    10:
        IF THIS^.WriteGCodeFile('TangentialCut.nc') THEN
            ADSLOGSTR(ADSLOG_MSGTYPE_HINT, 'Generator: Zapisano plik TangentialCut.nc', '');
            nBuildStep := 1000;
        END_IF

    1000:
        _Busy := FALSE;
        _Done := TRUE; 
        nBuildStep := 0;
        Build := TRUE;
        
END_CASE
END_METHOD

METHOD PROTECTED CalculateFootprint
VAR_INPUT
END_VAR
_NominalX := _Config.Diameter;
_NominalY := _Config.Diameter;
END_METHOD

PROPERTY ExecutionRoute : E_ExecutionRoute
GET
ExecutionRoute := E_ExecutionRoute.eGCode;
END_GET
END_PROPERTY

METHOD FB_init : BOOL
VAR_INPUT
	bInitRetains : BOOL; // if TRUE, the retain variables are initialized (warm start / cold start)
	bInCopyCode : BOOL;  // if TRUE, the instance afterwards gets moved into the copy code (online change)
END_VAR
_Limits.PanelFrontLength.MinVal := 100.0;
_Limits.PanelFrontLength.MaxVal := 2400.0;

_Limits.PanelFrontWidth.MinVal  := 100.0;
_Limits.PanelFrontWidth.MaxVal  := 1200.0;

_Limits.PanelHeight.MinVal      := 0.0;
_Limits.PanelHeight.MaxVal      := 0.0;

_Limits.RailHeightCorrection.MinVal := 0.0;
_Limits.RailHeightCorrection.MaxVal := 0.0;

_Limits.CuttingOverpass.MinVal := 0.0;
_Limits.CuttingOverpass.MaxVal := 50.0;

_Limits.GroovingOverpass.MinVal := 0.0;
_Limits.GroovingOverpass.MaxVal := 50.0;

_Limits.GrooveDepthZ.MinVal := 0.0;
_Limits.GrooveDepthZ.MaxVal := 9.0; 

_Limits.Diameter.MinVal := 10;
_Limits.Diameter.MaxVal := 600;
END_METHOD

END_FUNCTION_BLOCK

// ---- POUs/Builder/Recipes/FB_FeedRoundedRectangle.TcPOU
FUNCTION_BLOCK FB_FeedRoundedRectangle EXTENDS FB_RecipeBase

METHOD Build : BOOL
VAR
    TotalX, TotalY, Radius : LREAL;
    Velo : LREAL;
    localConfig : ST_GantryXYZ_Config;
	SmallRadius : LREAL;
    SmallMinX   : LREAL;
    SmallMaxX   : LREAL;
    SmallMinY   : LREAL;
    SmallMaxY   : LREAL;
END_VAR
_Busy := TRUE;
_Done := FALSE;
_Error := FALSE;
Build := FALSE;
THIS^.UpdateNestingLimits();

IF NOT _Config.IsValid THEN
    _Busy := FALSE;
    _Error := TRUE; 
    Build := FALSE;
    RETURN;
END_IF

// Gabaryty i promień
TotalX := _Config.PanelFrontWidth;
TotalY := _Config.PanelFrontLength;
Radius := _Config.Radius;

IF Radius > (TotalX / 2.0) THEN Radius := TotalX / 2.0; END_IF
IF Radius > (TotalY / 2.0) THEN Radius := TotalY / 2.0; END_IF

IF _ConfigProvider <> 0 THEN
    localConfig := _ConfigProvider.Config;
    Velo := localConfig.CuttingSpeedXY;
ELSE
    Velo := 50.0;
END_IF

// ===================================================
// DEFINICJA ILOŚCI I PUNKTÓW STARTOWYCH
// ===================================================
_ShapesCount := 1; 

// Kształt 1: Zewnętrzny prostokąt (100%) - Zaczynamy na środku PRAWEJ krawędzi
_ShapeStart[1].X := TotalX;
_ShapeStart[1].Y := TotalY / 2.0;

// Obliczenia dla małego prostokąta (50% wielkości, wyśrodkowany)
SmallMinX := TotalX * 0.25;
SmallMaxX := TotalX * 0.75;
SmallMinY := TotalY * 0.25;
SmallMaxY := TotalY * 0.75;
SmallRadius := Radius * 0.5;

// Kształt 2: Wewnętrzny prostokąt (50%) - Zaczynamy na środku PRAWEJ krawędzi
_ShapeStart[2].X := SmallMaxX;
_ShapeStart[2].Y := TotalY / 2.0;


// ============================================
// GENEROWANIE TABELI (Ruch CCW / Lewoskrętnie)
// ============================================
_GeometryWriter.Clear();
_GeometryWriter.EnableTangentialFollowing();

CASE _CurrentShapeIndex OF
    1:
        // ----------------------------------------------------
        // RYSOWANIE DUŻEGO PROSTOKĄTA (KSZTAŁT 1)
        // ----------------------------------------------------
        _GeometryWriter.AddStartPoint(_ShapeStart[1].X, _ShapeStart[1].Y);

        // 1. Prawa krawędź -> Prawy górny łuk (Tniemy w +Y, Q = 0)
        _GeometryWriter.AddLine(TotalX, TotalY - Radius, Velo);
        IF Radius > 0 THEN
            // FALSE = G03 = CounterClockwise (Lewoskrętnie)
            _GeometryWriter.AddArc(TotalX - Radius, TotalY, TotalX - Radius, TotalY - Radius, Velo, FALSE);
        END_IF

        // 2. Górna krawędź -> Lewy górny łuk (Tniemy w -X, Q = 90)
        _GeometryWriter.AddLine(Radius, TotalY, Velo);
        IF Radius > 0 THEN
            _GeometryWriter.AddArc(0.0, TotalY - Radius, Radius, TotalY - Radius, Velo, FALSE);
        END_IF

        // 3. Lewa krawędź -> Lewy dolny łuk (Tniemy w -Y, Q = 180)
        _GeometryWriter.AddLine(0.0, Radius, Velo);
        IF Radius > 0 THEN
            _GeometryWriter.AddArc(Radius, 0.0, Radius, Radius, Velo, FALSE);
        END_IF

        // 4. Dolna krawędź -> Prawy dolny łuk (Tniemy w +X, Q = 270)
        _GeometryWriter.AddLine(TotalX - Radius, 0.0, Velo);
        IF Radius > 0 THEN
            _GeometryWriter.AddArc(TotalX, Radius, TotalX - Radius, Radius, Velo, FALSE);
        END_IF

        // Zamknięcie na prawej krawędzi
        _GeometryWriter.AddLine(TotalX, TotalY / 2.0, Velo);

END_CASE

_GeometryWriter.EndTable();

_Busy := FALSE;
_Done := TRUE;
Build := TRUE;
END_METHOD

METHOD PROTECTED CalculateFootprint
VAR_INPUT
END_VAR
_NominalX := _Config.PanelFrontWidth;
_NominalY := _Config.PanelFrontLength;
END_METHOD

PROPERTY ExecutionRoute : E_ExecutionRoute
GET
ExecutionRoute := E_ExecutionRoute.eFeedTable;
END_GET
END_PROPERTY

METHOD FB_init : BOOL
VAR_INPUT
	bInitRetains : BOOL; // if TRUE, the retain variables are initialized (warm start / cold start)
	bInCopyCode : BOOL;  // if TRUE, the instance afterwards gets moved into the copy code (online change)
END_VAR
_Limits.PanelFrontLength.MinVal := 50.0;
_Limits.PanelFrontLength.MaxVal := 2400.0;

_Limits.PanelFrontWidth.MinVal  := 50.0;
_Limits.PanelFrontWidth.MaxVal  := 1200.0;

_Limits.PanelHeight.MinVal      := 0.0;
_Limits.PanelHeight.MaxVal      := 0.0;

_Limits.RailHeightCorrection.MinVal := 0.0;
_Limits.RailHeightCorrection.MaxVal := 0.0;

_Limits.CuttingOverpass.MinVal := 0.0;
_Limits.CuttingOverpass.MaxVal := 50.0;

_Limits.GroovingOverpass.MinVal := 0.0;
_Limits.GroovingOverpass.MaxVal := 50.0;

_Limits.GrooveDepthZ.MinVal := 0.0;
_Limits.GrooveDepthZ.MaxVal := 9.0; 

_Limits.CuttingOverpass.MinVal := 0.0;
_Limits.CuttingOverpass.MaxVal := 50.0;
_Limits.GroovingOverpass.MinVal := 0.0;
_Limits.GroovingOverpass.MaxVal := 50.0;

_Limits.Radius.MinVal := 10.0;     
_Limits.Radius.MaxVal := 600.0;
END_METHOD

END_FUNCTION_BLOCK

// ---- POUs/Builder/Recipes/FB_FeedCircle.TcPOU
FUNCTION_BLOCK FB_FeedCircle EXTENDS FB_RecipeBase

METHOD Build : BOOL
VAR
    TotalX, Radius : LREAL;
    Velo : LREAL;
    localConfig : ST_GantryXYZ_Config;
    LeadInY : LREAL := 20.0;
    LeadOutY : LREAL := 20.0;
END_VAR
_Busy := TRUE;
_Done := FALSE;
_Error := FALSE;
Build := FALSE;

THIS^.UpdateNestingLimits();

IF NOT _Config.IsValid THEN
    _Busy := FALSE;
    _Error := TRUE;
    RETURN;
END_IF

TotalX := _Config.Diameter;
Radius := TotalX / 2.0;

// ===================================================
// DEFINICJA ILOŚCI I PUNKTÓW STARTOWYCH
// ===================================================
_ShapesCount := 1; 

_ShapeStart[1].X := TotalX;
_ShapeStart[1].Y := Radius - LeadInY;

IF _ConfigProvider <> 0 THEN
    localConfig := _ConfigProvider.Config;
    Velo := localConfig.CuttingSpeedXY;
ELSE
    Velo := 50.0;
END_IF

_GeometryWriter.Clear();
_GeometryWriter.EnableTangentialFollowing();

// RYSOWANIE TYLKO TEGO KSZTAŁTU, O KTÓRY PROSI EXECUTOR
CASE _CurrentShapeIndex OF
    1:
        _GeometryWriter.AddStartPoint(_ShapeStart[1].X, _ShapeStart[1].Y); 
        _GeometryWriter.AddLine(TotalX, Radius, Velo); 
        _GeometryWriter.AddArc(0.0, Radius, Radius, Radius, Velo, FALSE);
        _GeometryWriter.AddArc(TotalX, Radius, Radius, Radius, Velo, FALSE);
        _GeometryWriter.AddLine(TotalX, Radius + LeadOutY, Velo); 
END_CASE

_GeometryWriter.EndTable();

_Busy := FALSE;
_Done := TRUE;
Build := TRUE;
END_METHOD

METHOD PROTECTED CalculateFootprint
VAR_INPUT
END_VAR
_NominalX := _Config.Diameter;
_NominalY := _Config.Diameter;
END_METHOD

PROPERTY ExecutionRoute : E_ExecutionRoute
GET
ExecutionRoute := E_ExecutionRoute.eFeedTable;
END_GET
END_PROPERTY

METHOD FB_init : BOOL
VAR_INPUT
	bInitRetains : BOOL; // if TRUE, the retain variables are initialized (warm start / cold start)
	bInCopyCode : BOOL;  // if TRUE, the instance afterwards gets moved into the copy code (online change)
END_VAR
_Limits.Diameter.MinVal := 50.0;
_Limits.Diameter.MaxVal := 1200.0;
_Limits.Radius.MinVal := 10.0;
_Limits.Radius.MaxVal := 100;

_Limits.CuttingOverpass.MinVal := 0.0;
_Limits.CuttingOverpass.MaxVal := 50.0;
_Limits.GroovingOverpass.MinVal := 0.0;
_Limits.GroovingOverpass.MaxVal := 50.0;
END_METHOD

END_FUNCTION_BLOCK

// ---- POUs/Builder/Recipes/FB_FeedMeina2_2000x1000.TcPOU
FUNCTION_BLOCK FB_FeedMeina2_2000x1000 EXTENDS FB_RecipeBase

METHOD Build : BOOL
VAR
    TotalX, TotalY, Radius : LREAL;
    Velo : LREAL;
    localConfig : ST_GantryXYZ_Config;
	
    // Zmienne do otworów
    HoleDistanceFromEdgeOfRail : LREAL := 100.0;
    SomeFixedDimension         : LREAL := 12.63;
    PanelRailOffsetX           : LREAL;
    PanelRailOffsetY           : LREAL;
    ExtrusionLengthX           : LREAL;
    ExtrusionLengthY           : LREAL;
    
    NumberOfHolesX             : INT := 3;
    NumberOfHolesY             : INT := 5;
    HolesSpacingX              : LREAL;
    HolesSpacingY              : LREAL;
    
    i                          : INT;
    holeIdx                    : INT;
	
	RailSlot  : LREAL := 29.0;
	BigSlot   : LREAL := 200.0;
	SmallSlot : LREAL := 100.0;

// Zmienne pomocnicze do generowania ścieżek
	sx : LREAL;
	sy : LREAL;
	dx : LREAL;
	dy : LREAL;
	r_val : LREAL;
	
END_VAR
_Busy := TRUE;
_Done := FALSE;
_Error := FALSE;
Build := FALSE;
THIS^.UpdateNestingLimits();

IF NOT _Config.IsValid THEN
    _Busy := FALSE;
    _Error := TRUE; 
    Build := FALSE;
    RETURN;
END_IF

// Gabaryty i promień
TotalX := 1000;
TotalY := 2000;
Radius := _Config.Radius;

IF Radius > (TotalX / 2.0) THEN Radius := TotalX / 2.0; END_IF
IF Radius > (TotalY / 2.0) THEN Radius := TotalY / 2.0; END_IF


// ===================================================
// OBLICZENIA DLA SZYN I OTWORÓW
// ===================================================
// Po poprawce: offset X uzależniony od X, a Y od Y
PanelRailOffsetX := 0.1 * TotalX;
PanelRailOffsetY := 0.1 * TotalY;

ExtrusionLengthX := TotalX - (2.0 * PanelRailOffsetX);
ExtrusionLengthY := TotalY - (2.0 * PanelRailOffsetY);

// Wyliczenie rozstawu (Zabezpieczenie przed dzieleniem przez zero, jeśli ktoś wpisze NumberOfHoles = 1)
IF NumberOfHolesX > 1 THEN
    HolesSpacingX := (ExtrusionLengthX - (2.0 * HoleDistanceFromEdgeOfRail)) / INT_TO_LREAL(NumberOfHolesX - 1);
ELSE
    HolesSpacingX := 0.0;
END_IF

IF NumberOfHolesY > 1 THEN
    HolesSpacingY := (ExtrusionLengthY - (2.0 * HoleDistanceFromEdgeOfRail)) / INT_TO_LREAL(NumberOfHolesY - 1);
ELSE
    HolesSpacingY := 0.0;
END_IF


// ===================================================
// GENEROWANIE OTWORÓW (Zoptymalizowana ścieżka po obwodzie)
// ===================================================
holeIdx := 1;

// 1. Otwór na dokładnym środku wycinanego detalu
_HolesDrill[holeIdx].X := LREAL_TO_REAL(TotalX / 2.0);
_HolesDrill[holeIdx].Y := LREAL_TO_REAL(TotalY / 2.0);

// 2. Rail Y1 (Lewa) - Ruch z GÓRY na DÓŁ
FOR i := NumberOfHolesY TO 1 BY -1 DO
    holeIdx := holeIdx + 1;
    _HolesDrill[holeIdx].X := LREAL_TO_REAL(PanelRailOffsetX - SomeFixedDimension);
    _HolesDrill[holeIdx].Y := LREAL_TO_REAL(PanelRailOffsetY + HoleDistanceFromEdgeOfRail + ((i - 1) * HolesSpacingY));
END_FOR

// 3. Rail X1 (Dolna) - Ruch z LEWEJ do PRAWEJ
FOR i := 1 TO NumberOfHolesX DO
    holeIdx := holeIdx + 1;
    _HolesDrill[holeIdx].X := LREAL_TO_REAL(PanelRailOffsetX + HoleDistanceFromEdgeOfRail + ((i - 1) * HolesSpacingX));
    _HolesDrill[holeIdx].Y := LREAL_TO_REAL(PanelRailOffsetY - SomeFixedDimension);
END_FOR

// 4. Rail Y2 (Prawa) - Ruch z DOŁU do GÓRY
FOR i := 1 TO NumberOfHolesY DO
    holeIdx := holeIdx + 1;
    _HolesDrill[holeIdx].X := LREAL_TO_REAL(PanelRailOffsetX + ExtrusionLengthX + SomeFixedDimension);
    _HolesDrill[holeIdx].Y := LREAL_TO_REAL(PanelRailOffsetY + HoleDistanceFromEdgeOfRail + ((i - 1) * HolesSpacingY));
END_FOR

// 5. Rail X2 (Górna) - Ruch z PRAWEJ do LEWEJ
FOR i := NumberOfHolesX TO 1 BY -1 DO
    holeIdx := holeIdx + 1;
    _HolesDrill[holeIdx].X := LREAL_TO_REAL(PanelRailOffsetX + HoleDistanceFromEdgeOfRail + ((i - 1) * HolesSpacingX));
    _HolesDrill[holeIdx].Y := LREAL_TO_REAL(PanelRailOffsetY + ExtrusionLengthY + SomeFixedDimension);
END_FOR

// Przypisanie całkowitej liczby otworów do recepty
_HolesToDrill := holeIdx;

// ===================================================
// DEFINICJA ILOŚCI I PUNKTÓW STARTOWYCH (Dla FeedTable)
// ===================================================
_ShapesCount := 6; // 1 główny panel + 5 nowych wycięć z tabeli

// 1. Kształt główny
_ShapeStart[1].X := 0.0;
_ShapeStart[1].Y := 0.0;

// 2. No. 1
_ShapeStart[2].X := 1030.0;
_ShapeStart[2].Y := 0.0;

// 3. No. 2
_ShapeStart[3].X := 1090.0;
_ShapeStart[3].Y := 0.0;

// 4. No. 3
_ShapeStart[4].X := 210.0;
_ShapeStart[4].Y := 2200.0;

// 5. No. 4
_ShapeStart[5].X := 410.0;
_ShapeStart[5].Y := 2150.0;

// 6. No. 5
_ShapeStart[6].X := 810.0;
_ShapeStart[6].Y := 2150.0;

IF _ConfigProvider <> 0 THEN
    localConfig := _ConfigProvider.Config;
    Velo := localConfig.CuttingSpeedXY;
ELSE
    Velo := 50.0;
END_IF

_GeometryWriter.Clear();
_GeometryWriter.EnableTangentialFollowing();

// Reset zmiennych pomocniczych przed każdym wywołaniem
sx := 0.0; sy := 0.0; dx := 0.0; dy := 0.0; r_val := 0.0;

// RYSOWANIE KSZTAŁTU ZGODNIE Z INDEKSEM
CASE _CurrentShapeIndex OF
    1:
        // ==========================================
        // KSZTAŁT 1 (Główny panel - Twój stary kod)
        // ==========================================
        _GeometryWriter.AddStartPoint(_ShapeStart[1].X, _ShapeStart[1].Y);

        _GeometryWriter.AddLine(0.0, TotalY - Radius, Velo);
        IF Radius > 0 THEN
            _GeometryWriter.AddArc(Radius, TotalY, Radius, TotalY - Radius, Velo, TRUE);
        END_IF

        _GeometryWriter.AddLine(TotalX - Radius, TotalY, Velo);
        IF Radius > 0 THEN
            _GeometryWriter.AddArc(TotalX, TotalY - Radius, TotalX - Radius, TotalY - Radius, Velo, TRUE);
        END_IF

        _GeometryWriter.AddLine(TotalX, Radius, Velo);
        IF Radius > 0 THEN
            _GeometryWriter.AddArc(TotalX - Radius, 0.0, TotalX - Radius, Radius, Velo, TRUE);
        END_IF

        _GeometryWriter.AddLine(Radius, 0.0, Velo);
        IF Radius > 0 THEN
            _GeometryWriter.AddArc(0.0, Radius, Radius, Radius, Velo, TRUE);
        END_IF

    2, 3, 4, 5, 6:
        // ==========================================
        // KSZTAŁTY OD 2 DO 6 (Z tabeli)
        // ==========================================
        // Przypisanie współrzędnych startowych dla aktualnego kształtu
        sx := _ShapeStart[_CurrentShapeIndex].X;
        sy := _ShapeStart[_CurrentShapeIndex].Y;
        r_val := 10.0; // Promień jest równy 10 dla wszystkich slotów

        // Dobór wymiarów na podstawie tego, który numer wycinamy
        IF _CurrentShapeIndex = 2 THEN
            dx := RailSlot;
            dy := ExtrusionLengthY;
        ELSIF _CurrentShapeIndex = 3 THEN
            dx := RailSlot;
            dy := ExtrusionLengthX;
        ELSIF _CurrentShapeIndex = 4 THEN
            dx := SmallSlot;
            dy := SmallSlot;
        ELSIF _CurrentShapeIndex = 5 THEN
            dx := BigSlot;
            dy := BigSlot;
        ELSIF _CurrentShapeIndex = 6 THEN
            dx := BigSlot;
            dy := BigSlot;
        END_IF

        // Wygenerowanie geometrycznej ścieżki (z absolutnym offsetem sx, sy)
        // Wkłuwamy się w lewym dolnym rogu (w odpad)
        _GeometryWriter.AddStartPoint(sx, sy);

        // 1. Lewa krawędź w górę
        _GeometryWriter.AddLine(sx, sy + dy - r_val, Velo);
        IF r_val > 0 THEN
            // Lewy górny łuk
            _GeometryWriter.AddArc(sx + r_val, sy + dy, sx + r_val, sy + dy - r_val, Velo, TRUE);
        END_IF

        // 2. Górna krawędź w prawo
        _GeometryWriter.AddLine(sx + dx - r_val, sy + dy, Velo);
        IF r_val > 0 THEN
            // Prawy górny łuk
            _GeometryWriter.AddArc(sx + dx, sy + dy - r_val, sx + dx - r_val, sy + dy - r_val, Velo, TRUE);
        END_IF

        // 3. Prawa krawędź w dół
        _GeometryWriter.AddLine(sx + dx, sy + r_val, Velo);
        IF r_val > 0 THEN
            // Prawy dolny łuk
            _GeometryWriter.AddArc(sx + dx - r_val, sy, sx + dx - r_val, sy + r_val, Velo, TRUE);
        END_IF

        // 4. Dolna krawędź w lewo i zamknięcie
        _GeometryWriter.AddLine(sx + r_val, sy, Velo);
        IF r_val > 0 THEN
            // Lewy dolny łuk
            _GeometryWriter.AddArc(sx, sy + r_val, sx + r_val, sy + r_val, Velo, TRUE);
        END_IF

END_CASE

_GeometryWriter.EndTable();

_Busy := FALSE;
_Done := TRUE;
Build := TRUE;
END_METHOD

METHOD PROTECTED CalculateFootprint
VAR_INPUT
END_VAR
_NominalX := 1200;
_NominalY := 2400;
END_METHOD

PROPERTY ExecutionRoute : E_ExecutionRoute
GET
ExecutionRoute := E_ExecutionRoute.eFeedTable;
END_GET
END_PROPERTY

METHOD FB_init : BOOL
VAR_INPUT
	bInitRetains : BOOL; // if TRUE, the retain variables are initialized (warm start / cold start)
	bInCopyCode : BOOL;  // if TRUE, the instance afterwards gets moved into the copy code (online change)
END_VAR
_Limits.PanelFrontLength.MinVal := 100.0;
_Limits.PanelFrontLength.MaxVal := 2400.0;

_Limits.PanelFrontWidth.MinVal  := 100.0;
_Limits.PanelFrontWidth.MaxVal  := 1200.0;

_Limits.PanelHeight.MinVal      := 0.0;
_Limits.PanelHeight.MaxVal      := 0.0;

_Limits.RailHeightCorrection.MinVal := 0.0;
_Limits.RailHeightCorrection.MaxVal := 0.0;

_Limits.CuttingOverpass.MinVal := 0.0;
_Limits.CuttingOverpass.MaxVal := 50.0;

_Limits.GroovingOverpass.MinVal := 0.0;
_Limits.GroovingOverpass.MaxVal := 50.0;

_Limits.GrooveDepthZ.MinVal := 0.0;
_Limits.GrooveDepthZ.MaxVal := 9.0; 

_Limits.CuttingOverpass.MinVal := 0.0;
_Limits.CuttingOverpass.MaxVal := 50.0;
_Limits.GroovingOverpass.MinVal := 0.0;
_Limits.GroovingOverpass.MaxVal := 50.0;

_Limits.Radius.MinVal := 10.0;     
_Limits.Radius.MaxVal := 600.0;
END_METHOD

END_FUNCTION_BLOCK

// ---- POUs/Builder/Recipes/FB_FeedMeina2_500x500.TcPOU
FUNCTION_BLOCK FB_FeedMeina2_500x500 EXTENDS FB_RecipeBase

METHOD Build : BOOL
VAR
    TotalX, TotalY, Radius : LREAL;
    Velo : LREAL;
    localConfig : ST_GantryXYZ_Config;
	
    // Zmienne do otworów
    HoleDistanceFromEdgeOfRail : LREAL := 100.0;
    SomeFixedDimension         : LREAL := 12.63;
    PanelRailOffsetX           : LREAL;
    PanelRailOffsetY           : LREAL;
    ExtrusionLengthX           : LREAL;
    ExtrusionLengthY           : LREAL;
    
    NumberOfHolesX             : INT := 3;
    NumberOfHolesY             : INT := 5;
    HolesSpacingX              : LREAL;
    HolesSpacingY              : LREAL;
    
    i                          : INT;
    holeIdx                    : INT;
	
	RailSlot  : LREAL := 29.0;
	BigSlot   : LREAL := 200.0;
	SmallSlot : LREAL := 100.0;

	PanelW : ARRAY[1..5] OF LREAL;
    PanelH : ARRAY[1..5] OF LREAL;
    PanelR : ARRAY[1..5] OF LREAL;
    X_Offset : LREAL;
    Y_Offset : LREAL;
    p : INT;

    // Stały wymiar szczelin ekstruzyjnych
    BaseExtrusion : LREAL;
	
	
// Zmienne pomocnicze do generowania ścieżek
	sx : LREAL;
	sy : LREAL;
	dx : LREAL;
	dy : LREAL;
	r_val : LREAL;
	
END_VAR
_Busy := TRUE;
_Done := FALSE;
_Error := FALSE;
Build := FALSE;
THIS^.UpdateNestingLimits();

IF NOT _Config.IsValid THEN
    _Busy := FALSE;
    _Error := TRUE; 
    Build := FALSE;
    RETURN;
END_IF

// ===================================================
// DEFINICJA PANELI GŁÓWNYCH (1 duży + 4 małe)
// ===================================================
// 1. Duży kwadrat (Oryginał)
_ShapeStart[1].X := 0.0;     _ShapeStart[1].Y := 0.0;
PanelW[1] := 1000.0;         PanelH[1] := 1000.0;
PanelR[1] := _Config.Radius; 

// 2. Mały kwadrat 1
_ShapeStart[2].X := 0.0;     _ShapeStart[2].Y := 1020.0;
PanelW[2] := 500.0;          PanelH[2] := 500.0;
PanelR[2] := 10.0;

// 3. Mały kwadrat 2
_ShapeStart[3].X := 0.0;     _ShapeStart[3].Y := 1540.0;
PanelW[3] := 500.0;          PanelH[3] := 500.0;
PanelR[3] := 10.0;

// 4. Mały kwadrat 3
_ShapeStart[4].X := 520.0;   _ShapeStart[4].Y := 1020.0;
PanelW[4] := 500.0;          PanelH[4] := 500.0;
PanelR[4] := 10.0;

// 5. Mały kwadrat 4
_ShapeStart[5].X := 520.0;   _ShapeStart[5].Y := 1540.0;
PanelW[5] := 500.0;          PanelH[5] := 500.0;
PanelR[5] := 10.0;

// ===================================================
// GENEROWANIE OTWORÓW DLA WSZYSTKICH 5 PANELI
// ===================================================
holeIdx := 0; 

FOR p := 1 TO 5 DO
    // Pobranie wymiarów dla aktualnie obliczanego panelu
    TotalX := PanelW[p];
    TotalY := PanelH[p];
    X_Offset := _ShapeStart[p].X;
    Y_Offset := _ShapeStart[p].Y;

    // Offsety i wyliczenia proporcjonalne do wymiarów konkretnego panelu
    PanelRailOffsetX := 0.1 * TotalX;
    PanelRailOffsetY := 0.1 * TotalY;

    ExtrusionLengthX := TotalX - (2.0 * PanelRailOffsetX);
    ExtrusionLengthY := TotalY - (2.0 * PanelRailOffsetY);

    IF NumberOfHolesX > 1 THEN
        HolesSpacingX := (ExtrusionLengthX - (2.0 * HoleDistanceFromEdgeOfRail)) / INT_TO_LREAL(NumberOfHolesX - 1);
    ELSE
        HolesSpacingX := 0.0;
    END_IF

    IF NumberOfHolesY > 1 THEN
        HolesSpacingY := (ExtrusionLengthY - (2.0 * HoleDistanceFromEdgeOfRail)) / INT_TO_LREAL(NumberOfHolesY - 1);
    ELSE
        HolesSpacingY := 0.0;
    END_IF

    // 1. Otwór na środku danego panelu
    holeIdx := holeIdx + 1;
    _HolesDrill[holeIdx].X := LREAL_TO_REAL((TotalX / 2.0) + X_Offset);
    _HolesDrill[holeIdx].Y := LREAL_TO_REAL((TotalY / 2.0) + Y_Offset);

    // 2. Rail Y1 (Lewa)
    FOR i := NumberOfHolesY TO 1 BY -1 DO
        holeIdx := holeIdx + 1;
        _HolesDrill[holeIdx].X := LREAL_TO_REAL(PanelRailOffsetX - SomeFixedDimension + X_Offset);
        _HolesDrill[holeIdx].Y := LREAL_TO_REAL(PanelRailOffsetY + HoleDistanceFromEdgeOfRail + ((i - 1) * HolesSpacingY) + Y_Offset);
    END_FOR

    // 3. Rail X1 (Dolna)
    FOR i := 1 TO NumberOfHolesX DO
        holeIdx := holeIdx + 1;
        _HolesDrill[holeIdx].X := LREAL_TO_REAL(PanelRailOffsetX + HoleDistanceFromEdgeOfRail + ((i - 1) * HolesSpacingX) + X_Offset);
        _HolesDrill[holeIdx].Y := LREAL_TO_REAL(PanelRailOffsetY - SomeFixedDimension + Y_Offset);
    END_FOR

    // 4. Rail Y2 (Prawa)
    FOR i := 1 TO NumberOfHolesY DO
        holeIdx := holeIdx + 1;
        _HolesDrill[holeIdx].X := LREAL_TO_REAL(PanelRailOffsetX + ExtrusionLengthX + SomeFixedDimension + X_Offset);
        _HolesDrill[holeIdx].Y := LREAL_TO_REAL(PanelRailOffsetY + HoleDistanceFromEdgeOfRail + ((i - 1) * HolesSpacingY) + Y_Offset);
    END_FOR

    // 5. Rail X2 (Górna)
    FOR i := NumberOfHolesX TO 1 BY -1 DO
        holeIdx := holeIdx + 1;
        _HolesDrill[holeIdx].X := LREAL_TO_REAL(PanelRailOffsetX + HoleDistanceFromEdgeOfRail + ((i - 1) * HolesSpacingX) + X_Offset);
        _HolesDrill[holeIdx].Y := LREAL_TO_REAL(PanelRailOffsetY + ExtrusionLengthY + SomeFixedDimension + Y_Offset);
    END_FOR
END_FOR

_HolesToDrill := holeIdx;

// ===================================================
// POZOSTAŁE WYCIĘCIA
// ===================================================
_ShapesCount := 10; // 5 paneli głównych + 5 małych wycięć

// No. 1 do No. 5 z poprzednich ustawień
_ShapeStart[6].X := 1030.0; _ShapeStart[6].Y := 0.0;
_ShapeStart[7].X := 1090.0; _ShapeStart[7].Y := 0.0;
_ShapeStart[8].X := 210.0;  _ShapeStart[8].Y := 2200.0;
_ShapeStart[9].X := 410.0;  _ShapeStart[9].Y := 2150.0;
_ShapeStart[10].X := 810.0; _ShapeStart[10].Y := 2150.0;

IF _ConfigProvider <> 0 THEN
    localConfig := _ConfigProvider.Config;
    Velo := localConfig.CuttingSpeedXY;
ELSE
    Velo := 50.0;
END_IF

_GeometryWriter.Clear();
_GeometryWriter.EnableTangentialFollowing();

sx := 0.0; sy := 0.0; dx := 0.0; dy := 0.0; r_val := 0.0;

// RYSOWANIE KSZTAŁTU ZGODNIE Z INDEKSEM
CASE _CurrentShapeIndex OF
    1, 2, 3, 4, 5:
        // ==========================================
        // RYSOWANIE PANELI (1 Duży + 4 Małe)
        // ==========================================
        sx := _ShapeStart[_CurrentShapeIndex].X;
        sy := _ShapeStart[_CurrentShapeIndex].Y;
        TotalX := PanelW[_CurrentShapeIndex];
        TotalY := PanelH[_CurrentShapeIndex];
        Radius := PanelR[_CurrentShapeIndex];

        IF Radius > (TotalX / 2.0) THEN Radius := TotalX / 2.0; END_IF
        IF Radius > (TotalY / 2.0) THEN Radius := TotalY / 2.0; END_IF

        _GeometryWriter.AddStartPoint(sx, sy);

        _GeometryWriter.AddLine(sx, sy + TotalY - Radius, Velo);
        IF Radius > 0 THEN
            _GeometryWriter.AddArc(sx + Radius, sy + TotalY, sx + Radius, sy + TotalY - Radius, Velo, TRUE);
        END_IF

        _GeometryWriter.AddLine(sx + TotalX - Radius, sy + TotalY, Velo);
        IF Radius > 0 THEN
            _GeometryWriter.AddArc(sx + TotalX, sy + TotalY - Radius, sx + TotalX - Radius, sy + TotalY - Radius, Velo, TRUE);
        END_IF

        _GeometryWriter.AddLine(sx + TotalX, sy + Radius, Velo);
        IF Radius > 0 THEN
            _GeometryWriter.AddArc(sx + TotalX - Radius, sy, sx + TotalX - Radius, sy + Radius, Velo, TRUE);
        END_IF

        _GeometryWriter.AddLine(sx + Radius, sy, Velo);
        IF Radius > 0 THEN
            _GeometryWriter.AddArc(sx, sy + Radius, sx + Radius, sy + Radius, Velo, TRUE);
        END_IF

    6, 7, 8, 9, 10:
        // ==========================================
        // RYSOWANIE WYCIĘĆ NA PROFILE
        // ==========================================
        sx := _ShapeStart[_CurrentShapeIndex].X;
        sy := _ShapeStart[_CurrentShapeIndex].Y;
        r_val := 10.0;

        // Stały wymiar dy/dx oparty na panelu 1000x1000: 1000 - 2*(10% z 1000) = 800
        BaseExtrusion := 800.0; 

        IF _CurrentShapeIndex = 6 THEN
            dx := RailSlot;
            dy := BaseExtrusion;
        ELSIF _CurrentShapeIndex = 7 THEN
            dx := RailSlot;
            dy := BaseExtrusion; 
        ELSIF _CurrentShapeIndex = 8 THEN
            dx := SmallSlot;
            dy := SmallSlot;
        ELSIF _CurrentShapeIndex = 9 THEN
            dx := BigSlot;
            dy := BigSlot;
        ELSIF _CurrentShapeIndex = 10 THEN
            dx := BigSlot;
            dy := BigSlot;
        END_IF

        _GeometryWriter.AddStartPoint(sx, sy);

        _GeometryWriter.AddLine(sx, sy + dy - r_val, Velo);
        IF r_val > 0 THEN
            _GeometryWriter.AddArc(sx + r_val, sy + dy, sx + r_val, sy + dy - r_val, Velo, TRUE);
        END_IF

        _GeometryWriter.AddLine(sx + dx - r_val, sy + dy, Velo);
        IF r_val > 0 THEN
            _GeometryWriter.AddArc(sx + dx, sy + dy - r_val, sx + dx - r_val, sy + dy - r_val, Velo, TRUE);
        END_IF

        _GeometryWriter.AddLine(sx + dx, sy + r_val, Velo);
        IF r_val > 0 THEN
            _GeometryWriter.AddArc(sx + dx - r_val, sy, sx + dx - r_val, sy + r_val, Velo, TRUE);
        END_IF

        _GeometryWriter.AddLine(sx + r_val, sy, Velo);
        IF r_val > 0 THEN
            _GeometryWriter.AddArc(sx, sy + r_val, sx + r_val, sy + r_val, Velo, TRUE);
        END_IF

END_CASE

_GeometryWriter.EndTable();

_Busy := FALSE;
_Done := TRUE;
Build := TRUE;
END_METHOD

METHOD PROTECTED CalculateFootprint
VAR_INPUT
END_VAR
_NominalX := 1200;
_NominalY := 2400;
END_METHOD

PROPERTY ExecutionRoute : E_ExecutionRoute
GET
ExecutionRoute := E_ExecutionRoute.ePTP;
END_GET
END_PROPERTY

METHOD FB_init : BOOL
VAR_INPUT
	bInitRetains : BOOL; // if TRUE, the retain variables are initialized (warm start / cold start)
	bInCopyCode : BOOL;  // if TRUE, the instance afterwards gets moved into the copy code (online change)
END_VAR
_Limits.PanelFrontLength.MinVal := 100.0;
_Limits.PanelFrontLength.MaxVal := 2400.0;

_Limits.PanelFrontWidth.MinVal  := 100.0;
_Limits.PanelFrontWidth.MaxVal  := 1200.0;

_Limits.PanelHeight.MinVal      := 0.0;
_Limits.PanelHeight.MaxVal      := 0.0;

_Limits.RailHeightCorrection.MinVal := 0.0;
_Limits.RailHeightCorrection.MaxVal := 0.0;

_Limits.CuttingOverpass.MinVal := 0.0;
_Limits.CuttingOverpass.MaxVal := 50.0;

_Limits.GroovingOverpass.MinVal := 0.0;
_Limits.GroovingOverpass.MaxVal := 50.0;

_Limits.GrooveDepthZ.MinVal := 0.0;
_Limits.GrooveDepthZ.MaxVal := 9.0; 

_Limits.CuttingOverpass.MinVal := 0.0;
_Limits.CuttingOverpass.MaxVal := 50.0;
_Limits.GroovingOverpass.MinVal := 0.0;
_Limits.GroovingOverpass.MaxVal := 50.0;

_Limits.Radius.MinVal := 10.0;     
_Limits.Radius.MaxVal := 600.0;
END_METHOD

END_FUNCTION_BLOCK

// ---- POUs/Builder/Recipes/FB_FeedMeina2_500x500_Circles.TcPOU
FUNCTION_BLOCK FB_FeedMeina2_500x500_Circles EXTENDS FB_RecipeBase

METHOD Build : BOOL
VAR
    TotalX, TotalY             : LREAL;
    CircleRadius               : LREAL;
    Velo                       : LREAL;
    localConfig                : ST_GantryXYZ_Config;
    
    X_Offset                   : LREAL; 
    Y_Offset                   : LREAL;
    p                          : INT;

    PanelW                     : ARRAY[1..10] OF LREAL; 
    PanelH                     : ARRAY[1..10] OF LREAL; 
    PanelX                     : ARRAY[1..10] OF LREAL; 
    PanelY                     : ARRAY[1..10] OF LREAL; 

    HoleDistanceFromEdgeOfRail : LREAL := 100.0;
    SomeFixedDimension         : LREAL := 12.63;
    PanelRailOffsetX           : LREAL;
    PanelRailOffsetY           : LREAL;
    ExtrusionLengthX           : LREAL;
    ExtrusionLengthY           : LREAL;
    BaseExtrusion              : LREAL; 
    
    NumberOfHolesX             : INT := 3;
    NumberOfHolesY             : INT := 5;
    HolesSpacingX              : LREAL;
    HolesSpacingY              : LREAL;
    
    i                          : INT;
    holeIdx                    : INT;
    
    RailSlot                   : LREAL := 29.0;
    BigSlot                    : LREAL := 200.0;
    SmallSlot                  : LREAL := 100.0;

    LeadInY                    : LREAL := 10.0;
    LeadOutY                   : LREAL := 10.0;

    sx                         : LREAL;
    sy                         : LREAL;
    dx                         : LREAL;
    dy                         : LREAL;
    r_val                      : LREAL;
END_VAR
_Busy := TRUE;
_Done := FALSE;
_Error := FALSE;
Build := FALSE;
THIS^.UpdateNestingLimits();

IF NOT _Config.IsValid THEN
    _Busy := FALSE;
    _Error := TRUE; 
    Build := FALSE;
    RETURN;
END_IF

PanelX[1] := 0.0;            PanelY[1] := 0.0;
PanelW[1] := 1000.0;         PanelH[1] := 1000.0;
_ShapeStart[1].X := PanelX[1] + PanelW[1];
_ShapeStart[1].Y := PanelY[1] + (PanelH[1] / 2.0) - LeadInY;

PanelX[2] := 0.0;            PanelY[2] := 1020.0;
PanelW[2] := 500.0;          PanelH[2] := 500.0;
_ShapeStart[2].X := PanelX[2] + PanelW[2];
_ShapeStart[2].Y := PanelY[2] + (PanelH[2] / 2.0) - LeadInY;

PanelX[3] := 0.0;            PanelY[3] := 1540.0;
PanelW[3] := 500.0;          PanelH[3] := 500.0;
_ShapeStart[3].X := PanelX[3] + PanelW[3];
_ShapeStart[3].Y := PanelY[3] + (PanelH[3] / 2.0) - LeadInY;

PanelX[4] := 520.0;          PanelY[4] := 1020.0;
PanelW[4] := 500.0;          PanelH[4] := 500.0;
_ShapeStart[4].X := PanelX[4] + PanelW[4];
_ShapeStart[4].Y := PanelY[4] + (PanelH[4] / 2.0) - LeadInY;

PanelX[5] := 520.0;          PanelY[5] := 1540.0;
PanelW[5] := 500.0;          PanelH[5] := 500.0;
_ShapeStart[5].X := PanelX[5] + PanelW[5];
_ShapeStart[5].Y := PanelY[5] + (PanelH[5] / 2.0) - LeadInY;

holeIdx := 0; 

FOR p := 1 TO 5 DO
    TotalX := PanelW[p];
    TotalY := PanelH[p];
    X_Offset := PanelX[p];
    Y_Offset := PanelY[p];

    PanelRailOffsetX := 0.1 * TotalX;
    PanelRailOffsetY := 0.1 * TotalY;

    ExtrusionLengthX := TotalX - (2.0 * PanelRailOffsetX);
    ExtrusionLengthY := TotalY - (2.0 * PanelRailOffsetY);

    IF NumberOfHolesX > 1 THEN
        HolesSpacingX := (ExtrusionLengthX - (2.0 * HoleDistanceFromEdgeOfRail)) / INT_TO_LREAL(NumberOfHolesX - 1);
    ELSE
        HolesSpacingX := 0.0;
    END_IF

    IF NumberOfHolesY > 1 THEN
        HolesSpacingY := (ExtrusionLengthY - (2.0 * HoleDistanceFromEdgeOfRail)) / INT_TO_LREAL(NumberOfHolesY - 1);
    ELSE
        HolesSpacingY := 0.0;
    END_IF

    holeIdx := holeIdx + 1;
    _HolesDrill[holeIdx].X := LREAL_TO_REAL((TotalX / 2.0) + X_Offset);
    _HolesDrill[holeIdx].Y := LREAL_TO_REAL((TotalY / 2.0) + Y_Offset);

    FOR i := NumberOfHolesY TO 1 BY -1 DO
        holeIdx := holeIdx + 1;
        _HolesDrill[holeIdx].X := LREAL_TO_REAL(PanelRailOffsetX - SomeFixedDimension + X_Offset);
        _HolesDrill[holeIdx].Y := LREAL_TO_REAL(PanelRailOffsetY + HoleDistanceFromEdgeOfRail + ((i - 1) * HolesSpacingY) + Y_Offset);
    END_FOR

    FOR i := 1 TO NumberOfHolesX DO
        holeIdx := holeIdx + 1;
        _HolesDrill[holeIdx].X := LREAL_TO_REAL(PanelRailOffsetX + HoleDistanceFromEdgeOfRail + ((i - 1) * HolesSpacingX) + X_Offset);
        _HolesDrill[holeIdx].Y := LREAL_TO_REAL(PanelRailOffsetY - SomeFixedDimension + Y_Offset);
    END_FOR

    FOR i := 1 TO NumberOfHolesY DO
        holeIdx := holeIdx + 1;
        _HolesDrill[holeIdx].X := LREAL_TO_REAL(PanelRailOffsetX + ExtrusionLengthX + SomeFixedDimension + X_Offset);
        _HolesDrill[holeIdx].Y := LREAL_TO_REAL(PanelRailOffsetY + HoleDistanceFromEdgeOfRail + ((i - 1) * HolesSpacingY) + Y_Offset);
    END_FOR

    FOR i := NumberOfHolesX TO 1 BY -1 DO
        holeIdx := holeIdx + 1;
        _HolesDrill[holeIdx].X := LREAL_TO_REAL(PanelRailOffsetX + HoleDistanceFromEdgeOfRail + ((i - 1) * HolesSpacingX) + X_Offset);
        _HolesDrill[holeIdx].Y := LREAL_TO_REAL(PanelRailOffsetY + ExtrusionLengthY + SomeFixedDimension + Y_Offset);
    END_FOR
END_FOR

_HolesToDrill := holeIdx;

_ShapesCount := 10; 

_ShapeStart[6].X := 1030.0; _ShapeStart[6].Y := 0.0;
_ShapeStart[7].X := 1090.0; _ShapeStart[7].Y := 0.0;
_ShapeStart[8].X := 210.0;  _ShapeStart[8].Y := 2200.0;
_ShapeStart[9].X := 410.0;  _ShapeStart[9].Y := 2150.0;
_ShapeStart[10].X := 810.0; _ShapeStart[10].Y := 2150.0;

IF _ConfigProvider <> 0 THEN
    localConfig := _ConfigProvider.Config;
    Velo := localConfig.CuttingSpeedXY;
ELSE
    Velo := 50.0;
END_IF

_GeometryWriter.Clear();
_GeometryWriter.EnableTangentialFollowing();

sx := 0.0; sy := 0.0; dx := 0.0; dy := 0.0; r_val := 0.0;

CASE _CurrentShapeIndex OF
    1, 2, 3, 4, 5:
        sx := PanelX[_CurrentShapeIndex];
        sy := PanelY[_CurrentShapeIndex];
        TotalX := PanelW[_CurrentShapeIndex];
        TotalY := PanelH[_CurrentShapeIndex];
        CircleRadius := TotalX / 2.0;

        _GeometryWriter.AddStartPoint(_ShapeStart[_CurrentShapeIndex].X, _ShapeStart[_CurrentShapeIndex].Y); 
        
        _GeometryWriter.AddLine(sx + TotalX, sy + CircleRadius, Velo); 
        
        _GeometryWriter.AddArc(sx, sy + CircleRadius, sx + CircleRadius, sy + CircleRadius, Velo, FALSE);
        
        _GeometryWriter.AddArc(sx + TotalX, sy + CircleRadius, sx + CircleRadius, sy + CircleRadius, Velo, FALSE);
        
        _GeometryWriter.AddLine(sx + TotalX, sy + CircleRadius + LeadOutY, Velo); 

    6, 7, 8, 9, 10:
        sx := _ShapeStart[_CurrentShapeIndex].X;
        sy := _ShapeStart[_CurrentShapeIndex].Y;
        r_val := 10.0;

        BaseExtrusion := 800.0; 

        IF _CurrentShapeIndex = 6 THEN
            dx := RailSlot;
            dy := BaseExtrusion;
        ELSIF _CurrentShapeIndex = 7 THEN
            dx := RailSlot;
            dy := BaseExtrusion; 
        ELSIF _CurrentShapeIndex = 8 THEN
            dx := SmallSlot;
            dy := SmallSlot;
        ELSIF _CurrentShapeIndex = 9 THEN
            dx := BigSlot;
            dy := BigSlot;
        ELSIF _CurrentShapeIndex = 10 THEN
            dx := BigSlot;
            dy := BigSlot;
        END_IF

        _GeometryWriter.AddStartPoint(sx, sy);

        _GeometryWriter.AddLine(sx, sy + dy - r_val, Velo);
        IF r_val > 0 THEN
            _GeometryWriter.AddArc(sx + r_val, sy + dy, sx + r_val, sy + dy - r_val, Velo, TRUE);
        END_IF

        _GeometryWriter.AddLine(sx + dx - r_val, sy + dy, Velo);
        IF r_val > 0 THEN
            _GeometryWriter.AddArc(sx + dx, sy + dy - r_val, sx + dx - r_val, sy + dy - r_val, Velo, TRUE);
        END_IF

        _GeometryWriter.AddLine(sx + dx, sy + r_val, Velo);
        IF r_val > 0 THEN
            _GeometryWriter.AddArc(sx + dx - r_val, sy, sx + dx - r_val, sy + r_val, Velo, TRUE);
        END_IF

        _GeometryWriter.AddLine(sx + r_val, sy, Velo);
        IF r_val > 0 THEN
            _GeometryWriter.AddArc(sx, sy + r_val, sx + r_val, sy + r_val, Velo, TRUE);
        END_IF

END_CASE

_GeometryWriter.EndTable();

_Busy := FALSE;
_Done := TRUE;
Build := TRUE;
END_METHOD

METHOD PROTECTED CalculateFootprint
VAR_INPUT
END_VAR
_NominalX := 1200;
_NominalY := 2400;
END_METHOD

PROPERTY ExecutionRoute : E_ExecutionRoute
GET
ExecutionRoute := E_ExecutionRoute.eFeedTable;
END_GET
END_PROPERTY

METHOD FB_init : BOOL
VAR_INPUT
	bInitRetains : BOOL; // if TRUE, the retain variables are initialized (warm start / cold start)
	bInCopyCode : BOOL;  // if TRUE, the instance afterwards gets moved into the copy code (online change)
END_VAR
_Limits.PanelFrontLength.MinVal := 100.0;
_Limits.PanelFrontLength.MaxVal := 2400.0;

_Limits.PanelFrontWidth.MinVal  := 100.0;
_Limits.PanelFrontWidth.MaxVal  := 1200.0;

_Limits.PanelHeight.MinVal      := 0.0;
_Limits.PanelHeight.MaxVal      := 0.0;

_Limits.RailHeightCorrection.MinVal := 0.0;
_Limits.RailHeightCorrection.MaxVal := 0.0;

_Limits.CuttingOverpass.MinVal := 0.0;
_Limits.CuttingOverpass.MaxVal := 50.0;

_Limits.GroovingOverpass.MinVal := 0.0;
_Limits.GroovingOverpass.MaxVal := 50.0;

_Limits.GrooveDepthZ.MinVal := 0.0;
_Limits.GrooveDepthZ.MaxVal := 9.0; 

_Limits.CuttingOverpass.MinVal := 0.0;
_Limits.CuttingOverpass.MaxVal := 50.0;
_Limits.GroovingOverpass.MinVal := 0.0;
_Limits.GroovingOverpass.MaxVal := 50.0;

_Limits.Radius.MinVal := 10.0;     
_Limits.Radius.MaxVal := 600.0;
END_METHOD

END_FUNCTION_BLOCK

// ---- POUs/Builder/Recipes/FB_FeedMeina2_750x750.TcPOU
FUNCTION_BLOCK FB_FeedMeina2_750x750 EXTENDS FB_RecipeBase

METHOD Build : BOOL
VAR
    TotalX, TotalY, Radius : LREAL;
    CircleRadius           : LREAL;
    Velo                   : LREAL;
    localConfig            : ST_GantryXYZ_Config;
    
    PanelGap               : LREAL;
    Y_Offset               : LREAL;
    p                      : INT;

    HoleDistanceFromEdgeOfRail : LREAL := 100.0;
    SomeFixedDimension         : LREAL := 12.63;
    PanelRailOffsetX           : LREAL;
    PanelRailOffsetY           : LREAL;
    ExtrusionLengthX           : LREAL;
    ExtrusionLengthY           : LREAL;
    
    NumberOfHolesX             : INT := 3;
    NumberOfHolesY             : INT := 5;
    HolesSpacingX              : LREAL;
    HolesSpacingY              : LREAL;
    
    i                          : INT;
    holeIdx                    : INT;
    
    RailSlot  : LREAL := 29.0;
    BigSlot   : LREAL := 200.0;
    SmallSlot : LREAL := 100.0;

    LeadInY   : LREAL := 10.0;
    LeadOutY  : LREAL := 10.0;

    sx : LREAL;
    sy : LREAL;
    dx : LREAL;
    dy : LREAL;
    r_val : LREAL;
END_VAR
_Busy := TRUE;
_Done := FALSE;
_Error := FALSE;
Build := FALSE;
THIS^.UpdateNestingLimits();

IF NOT _Config.IsValid THEN
    _Busy := FALSE;
    _Error := TRUE; 
    Build := FALSE;
    RETURN;
END_IF

// ===================================================
// NOWE GEOMETRIE DLA TRZECH KWADRATÓW 750x750
// ===================================================
TotalX := 750.0; 
TotalY := 750.0; 
Radius := _Config.Radius;

IF Radius > (TotalX / 2.0) THEN Radius := TotalX / 2.0; END_IF
IF Radius > (TotalY / 2.0) THEN Radius := TotalY / 2.0; END_IF

// Przerwa między panelami (20 mm) w osi Y
PanelGap := 20.0; 

// Offsety dla szyn
PanelRailOffsetX := 0.1 * TotalX;
PanelRailOffsetY := 0.1 * TotalY;

ExtrusionLengthX := TotalX - (2.0 * PanelRailOffsetX);
ExtrusionLengthY := TotalY - (2.0 * PanelRailOffsetY);

// Wyliczenie rozstawu otworów
IF NumberOfHolesX > 1 THEN
    HolesSpacingX := (ExtrusionLengthX - (2.0 * HoleDistanceFromEdgeOfRail)) / INT_TO_LREAL(NumberOfHolesX - 1);
ELSE
    HolesSpacingX := 0.0;
END_IF

IF NumberOfHolesY > 1 THEN
    HolesSpacingY := (ExtrusionLengthY - (2.0 * HoleDistanceFromEdgeOfRail)) / INT_TO_LREAL(NumberOfHolesY - 1);
ELSE
    HolesSpacingY := 0.0;
END_IF


// ===================================================
// GENEROWANIE OTWORÓW DLA TRZECH PANELÓW
// ===================================================
holeIdx := 0; 

// Pętla dla 3 paneli: 0, 1, 2
FOR p := 0 TO 2 DO
    Y_Offset := INT_TO_LREAL(p) * (TotalY + PanelGap);

    // 1. Otwór na dokładnym środku danego panelu
    holeIdx := holeIdx + 1;
    _HolesDrill[holeIdx].X := LREAL_TO_REAL(TotalX / 2.0);
    _HolesDrill[holeIdx].Y := LREAL_TO_REAL((TotalY / 2.0) + Y_Offset);

    // 2. Rail Y1 (Lewa)
    FOR i := NumberOfHolesY TO 1 BY -1 DO
        holeIdx := holeIdx + 1;
        _HolesDrill[holeIdx].X := LREAL_TO_REAL(PanelRailOffsetX - SomeFixedDimension);
        _HolesDrill[holeIdx].Y := LREAL_TO_REAL(PanelRailOffsetY + HoleDistanceFromEdgeOfRail + ((i - 1) * HolesSpacingY) + Y_Offset);
    END_FOR

    // 3. Rail X1 (Dolna)
    FOR i := 1 TO NumberOfHolesX DO
        holeIdx := holeIdx + 1;
        _HolesDrill[holeIdx].X := LREAL_TO_REAL(PanelRailOffsetX + HoleDistanceFromEdgeOfRail + ((i - 1) * HolesSpacingX));
        _HolesDrill[holeIdx].Y := LREAL_TO_REAL(PanelRailOffsetY - SomeFixedDimension + Y_Offset);
    END_FOR

    // 4. Rail Y2 (Prawa)
    FOR i := 1 TO NumberOfHolesY DO
        holeIdx := holeIdx + 1;
        _HolesDrill[holeIdx].X := LREAL_TO_REAL(PanelRailOffsetX + ExtrusionLengthX + SomeFixedDimension);
        _HolesDrill[holeIdx].Y := LREAL_TO_REAL(PanelRailOffsetY + HoleDistanceFromEdgeOfRail + ((i - 1) * HolesSpacingY) + Y_Offset);
    END_FOR

    // 5. Rail X2 (Górna)
    FOR i := NumberOfHolesX TO 1 BY -1 DO
        holeIdx := holeIdx + 1;
        _HolesDrill[holeIdx].X := LREAL_TO_REAL(PanelRailOffsetX + HoleDistanceFromEdgeOfRail + ((i - 1) * HolesSpacingX));
        _HolesDrill[holeIdx].Y := LREAL_TO_REAL(PanelRailOffsetY + ExtrusionLengthY + SomeFixedDimension + Y_Offset);
    END_FOR
END_FOR

_HolesToDrill := holeIdx;

// ===================================================
// DEFINICJA ILOŚCI I PUNKTÓW STARTOWYCH
// ===================================================
_ShapesCount := 8;

// 1. Kształt główny - Panel Dolny
_ShapeStart[1].X := 0.0;
_ShapeStart[1].Y := 0.0;

// 2. Kształt główny - Panel Środkowy
_ShapeStart[2].X := 0.0;
_ShapeStart[2].Y := TotalY + PanelGap; // offset 770.0

// 3. Kształt główny - Panel Górny
_ShapeStart[3].X := 0.0;
_ShapeStart[3].Y := 2.0 * (TotalY + PanelGap); // offset 1540.0

// ===================================================
// WSPÓŁRZĘDNE SLOTÓW PRZYWRÓCONE Z PIERWSZEGO PROGRAMU
// ===================================================
_ShapeStart[4].X := 900.0;
_ShapeStart[4].Y := 125.0;

_ShapeStart[5].X := 900.0;
_ShapeStart[5].Y := 875.0;

_ShapeStart[6].X := 870.0;
_ShapeStart[6].Y := 520.0;

_ShapeStart[7].X := 870.0;
_ShapeStart[7].Y := 220.0;

_ShapeStart[8].X := 920.0;
_ShapeStart[8].Y := 20.0;


IF _ConfigProvider <> 0 THEN
    localConfig := _ConfigProvider.Config;
    Velo := localConfig.CuttingSpeedXY;
ELSE
    Velo := 50.0;
END_IF

_GeometryWriter.Clear();
_GeometryWriter.EnableTangentialFollowing();

sx := 0.0; sy := 0.0; dx := 0.0; dy := 0.0; r_val := 0.0;

// RYSOWANIE KSZTAŁTU ZGODNIE Z INDEKSEM
CASE _CurrentShapeIndex OF
    
    // Cięcie trzech paneli (kwadratów)
    1, 2, 3:
        sx := _ShapeStart[_CurrentShapeIndex].X;
        sy := _ShapeStart[_CurrentShapeIndex].Y;

        _GeometryWriter.AddStartPoint(sx, sy);

        _GeometryWriter.AddLine(sx, sy + TotalY - Radius, Velo);
        IF Radius > 0 THEN
            _GeometryWriter.AddArc(sx + Radius, sy + TotalY, sx + Radius, sy + TotalY - Radius, Velo, TRUE);
        END_IF

        _GeometryWriter.AddLine(sx + TotalX - Radius, sy + TotalY, Velo);
        IF Radius > 0 THEN
            _GeometryWriter.AddArc(sx + TotalX, sy + TotalY - Radius, sx + TotalX - Radius, sy + TotalY - Radius, Velo, TRUE);
        END_IF

        _GeometryWriter.AddLine(sx + TotalX, sy + Radius, Velo);
        IF Radius > 0 THEN
            _GeometryWriter.AddArc(sx + TotalX - Radius, sy, sx + TotalX - Radius, sy + Radius, Velo, TRUE);
        END_IF

        _GeometryWriter.AddLine(sx + Radius, sy, Velo);
        IF Radius > 0 THEN
            _GeometryWriter.AddArc(sx, sy + Radius, sx + Radius, sy + Radius, Velo, TRUE);
        END_IF

    // Wycięcia wewnętrzne z odpowiednio przypisaną logiką
    4, 5, 6, 7, 8:
        sx := _ShapeStart[_CurrentShapeIndex].X;
        sy := _ShapeStart[_CurrentShapeIndex].Y;
        r_val := 10.0;

        IF _CurrentShapeIndex = 4 THEN
            dx := RailSlot;
            dy := ExtrusionLengthY;
        ELSIF _CurrentShapeIndex = 5 THEN
            dx := RailSlot;
            dy := ExtrusionLengthX; 
        ELSIF _CurrentShapeIndex = 6 THEN
            dx := SmallSlot;
            dy := SmallSlot;
        ELSIF _CurrentShapeIndex = 7 THEN
            dx := BigSlot;
            dy := BigSlot;
        ELSIF _CurrentShapeIndex = 8 THEN
            dx := BigSlot;
            dy := BigSlot;
        END_IF

        _GeometryWriter.AddStartPoint(sx, sy);

        _GeometryWriter.AddLine(sx, sy + dy - r_val, Velo);
        IF r_val > 0 THEN
            _GeometryWriter.AddArc(sx + r_val, sy + dy, sx + r_val, sy + dy - r_val, Velo, TRUE);
        END_IF

        _GeometryWriter.AddLine(sx + dx - r_val, sy + dy, Velo);
        IF r_val > 0 THEN
            _GeometryWriter.AddArc(sx + dx, sy + dy - r_val, sx + dx - r_val, sy + dy - r_val, Velo, TRUE);
        END_IF

        _GeometryWriter.AddLine(sx + dx, sy + r_val, Velo);
        IF r_val > 0 THEN
            _GeometryWriter.AddArc(sx + dx - r_val, sy, sx + dx - r_val, sy + r_val, Velo, TRUE);
        END_IF

        _GeometryWriter.AddLine(sx + r_val, sy, Velo);
        IF r_val > 0 THEN
            _GeometryWriter.AddArc(sx, sy + r_val, sx + r_val, sy + r_val, Velo, TRUE);
        END_IF

END_CASE

_GeometryWriter.EndTable();

_Busy := FALSE;
_Done := TRUE;
Build := TRUE;
END_METHOD

METHOD PROTECTED CalculateFootprint
VAR_INPUT
END_VAR
_NominalX := 1200;
_NominalY := 2400;
END_METHOD

PROPERTY ExecutionRoute : E_ExecutionRoute
GET
ExecutionRoute := E_ExecutionRoute.eFeedTable;
END_GET
END_PROPERTY

METHOD FB_init : BOOL
VAR_INPUT
	bInitRetains : BOOL; // if TRUE, the retain variables are initialized (warm start / cold start)
	bInCopyCode : BOOL;  // if TRUE, the instance afterwards gets moved into the copy code (online change)
END_VAR
_Limits.PanelFrontLength.MinVal := 100.0;
_Limits.PanelFrontLength.MaxVal := 2400.0;

_Limits.PanelFrontWidth.MinVal  := 100.0;
_Limits.PanelFrontWidth.MaxVal  := 1200.0;

_Limits.PanelHeight.MinVal      := 0.0;
_Limits.PanelHeight.MaxVal      := 0.0;

_Limits.RailHeightCorrection.MinVal := 0.0;
_Limits.RailHeightCorrection.MaxVal := 0.0;

_Limits.CuttingOverpass.MinVal := 0.0;
_Limits.CuttingOverpass.MaxVal := 50.0;

_Limits.GroovingOverpass.MinVal := 0.0;
_Limits.GroovingOverpass.MaxVal := 50.0;

_Limits.GrooveDepthZ.MinVal := 0.0;
_Limits.GrooveDepthZ.MaxVal := 9.0; 

_Limits.CuttingOverpass.MinVal := 0.0;
_Limits.CuttingOverpass.MaxVal := 50.0;
_Limits.GroovingOverpass.MinVal := 0.0;
_Limits.GroovingOverpass.MaxVal := 50.0;

_Limits.Radius.MinVal := 10.0;     
_Limits.Radius.MaxVal := 600.0;
END_METHOD

END_FUNCTION_BLOCK

// ---- POUs/Builder/Recipes/FB_FeedMeina2_750x750_Circles.TcPOU
FUNCTION_BLOCK FB_FeedMeina2_750x750_Circles EXTENDS FB_RecipeBase

METHOD Build : BOOL
VAR
    TotalX, TotalY, Radius : LREAL;
    CircleRadius           : LREAL;
    Velo                   : LREAL;
    localConfig            : ST_GantryXYZ_Config;
    
    PanelGap               : LREAL;
    Y_Offset               : LREAL;
    p                      : INT;

    HoleDistanceFromEdgeOfRail : LREAL := 100.0;
    SomeFixedDimension         : LREAL := 12.63;
    PanelRailOffsetX           : LREAL;
    PanelRailOffsetY           : LREAL;
    ExtrusionLengthX           : LREAL;
    ExtrusionLengthY           : LREAL;
    
    NumberOfHolesX             : INT := 3;
    NumberOfHolesY             : INT := 5;
    HolesSpacingX              : LREAL;
    HolesSpacingY              : LREAL;
    
    i                          : INT;
    holeIdx                    : INT;
    
    RailSlot  : LREAL := 29.0;
    BigSlot   : LREAL := 200.0;
    SmallSlot : LREAL := 100.0;

    LeadInY   : LREAL := 10.0;
    LeadOutY  : LREAL := 10.0;

    sx : LREAL;
    sy : LREAL;
    dx : LREAL;
    dy : LREAL;
    r_val : LREAL;
END_VAR
_Busy := TRUE;
_Done := FALSE;
_Error := FALSE;
Build := FALSE;
THIS^.UpdateNestingLimits();

IF NOT _Config.IsValid THEN
    _Busy := FALSE;
    _Error := TRUE; 
    Build := FALSE;
    RETURN;
END_IF

// Zmiana rozmiaru na 750mm
TotalX := 750.0;
TotalY := 750.0;
CircleRadius := TotalX / 2.0;

PanelGap := 20.0; 

PanelRailOffsetX := 0.1 * TotalX;
PanelRailOffsetY := 0.1 * TotalY;

ExtrusionLengthX := TotalX - (2.0 * PanelRailOffsetX);
ExtrusionLengthY := TotalY - (2.0 * PanelRailOffsetY);

IF NumberOfHolesX > 1 THEN
    HolesSpacingX := (ExtrusionLengthX - (2.0 * HoleDistanceFromEdgeOfRail)) / INT_TO_LREAL(NumberOfHolesX - 1);
ELSE
    HolesSpacingX := 0.0;
END_IF

IF NumberOfHolesY > 1 THEN
    HolesSpacingY := (ExtrusionLengthY - (2.0 * HoleDistanceFromEdgeOfRail)) / INT_TO_LREAL(NumberOfHolesY - 1);
ELSE
    HolesSpacingY := 0.0;
END_IF

holeIdx := 0; 

// Pętla zmieniona na 3 elementy (0 DO 2)
FOR p := 0 TO 2 DO
    Y_Offset := INT_TO_LREAL(p) * (TotalY + PanelGap);

    holeIdx := holeIdx + 1;
    _HolesDrill[holeIdx].X := LREAL_TO_REAL(TotalX / 2.0);
    _HolesDrill[holeIdx].Y := LREAL_TO_REAL((TotalY / 2.0) + Y_Offset);

    FOR i := NumberOfHolesY TO 1 BY -1 DO
        holeIdx := holeIdx + 1;
        _HolesDrill[holeIdx].X := LREAL_TO_REAL(PanelRailOffsetX - SomeFixedDimension);
        _HolesDrill[holeIdx].Y := LREAL_TO_REAL(PanelRailOffsetY + HoleDistanceFromEdgeOfRail + ((i - 1) * HolesSpacingY) + Y_Offset);
    END_FOR

    FOR i := 1 TO NumberOfHolesX DO
        holeIdx := holeIdx + 1;
        _HolesDrill[holeIdx].X := LREAL_TO_REAL(PanelRailOffsetX + HoleDistanceFromEdgeOfRail + ((i - 1) * HolesSpacingX));
        _HolesDrill[holeIdx].Y := LREAL_TO_REAL(PanelRailOffsetY - SomeFixedDimension + Y_Offset);
    END_FOR

    FOR i := 1 TO NumberOfHolesY DO
        holeIdx := holeIdx + 1;
        _HolesDrill[holeIdx].X := LREAL_TO_REAL(PanelRailOffsetX + ExtrusionLengthX + SomeFixedDimension);
        _HolesDrill[holeIdx].Y := LREAL_TO_REAL(PanelRailOffsetY + HoleDistanceFromEdgeOfRail + ((i - 1) * HolesSpacingY) + Y_Offset);
    END_FOR

    FOR i := NumberOfHolesX TO 1 BY -1 DO
        holeIdx := holeIdx + 1;
        _HolesDrill[holeIdx].X := LREAL_TO_REAL(PanelRailOffsetX + HoleDistanceFromEdgeOfRail + ((i - 1) * HolesSpacingX));
        _HolesDrill[holeIdx].Y := LREAL_TO_REAL(PanelRailOffsetY + ExtrusionLengthY + SomeFixedDimension + Y_Offset);
    END_FOR
END_FOR

_HolesToDrill := holeIdx;

// Liczba kształtów to teraz 8 (3 kółka + 5 dotychczasowych profili/otworów)
_ShapesCount := 8; 

// Kółko 1
_ShapeStart[1].X := TotalX;
_ShapeStart[1].Y := CircleRadius - LeadInY;

// Kółko 2
_ShapeStart[2].X := TotalX;
_ShapeStart[2].Y := TotalY + PanelGap + CircleRadius - LeadInY;

// Kółko 3
_ShapeStart[3].X := TotalX;
_ShapeStart[3].Y := 2.0 * (TotalY + PanelGap) + CircleRadius - LeadInY;

// Pozostałe kształty przesunięte na indeksy 4-8 
// UWAGA: Stałe współrzędne > 750 (np. 900.0) mogą wymagać Twojej poprawki do nowego wymiaru TotalX/Y
_ShapeStart[4].X := 900.0;
_ShapeStart[4].Y := 125.0;

_ShapeStart[5].X := 900.0;
_ShapeStart[5].Y := 875.0;

_ShapeStart[6].X := 920.0;
_ShapeStart[6].Y := 20.0;

_ShapeStart[7].X := 870.0;
_ShapeStart[7].Y := 220.0;

_ShapeStart[8].X := 870.0;
_ShapeStart[8].Y := 520.0;

IF _ConfigProvider <> 0 THEN
    localConfig := _ConfigProvider.Config;
    Velo := localConfig.CuttingSpeedXY;
ELSE
    Velo := 50.0;
END_IF

_GeometryWriter.Clear();
_GeometryWriter.EnableTangentialFollowing();

sx := 0.0; sy := 0.0; dx := 0.0; dy := 0.0; r_val := 0.0;

CASE _CurrentShapeIndex OF
    // Obsługa cięcia 3 kółek w ten sam sposób
    1, 2, 3:
        Y_Offset := INT_TO_LREAL(_CurrentShapeIndex - 1) * (TotalY + PanelGap);

        _GeometryWriter.AddStartPoint(_ShapeStart[_CurrentShapeIndex].X, _ShapeStart[_CurrentShapeIndex].Y); 
        _GeometryWriter.AddLine(TotalX, CircleRadius + Y_Offset, Velo); 
        _GeometryWriter.AddArc(0.0, CircleRadius + Y_Offset, CircleRadius, CircleRadius + Y_Offset, Velo, FALSE);
        _GeometryWriter.AddArc(TotalX, CircleRadius + Y_Offset, CircleRadius, CircleRadius + Y_Offset, Velo, FALSE);
        _GeometryWriter.AddLine(TotalX, CircleRadius + LeadOutY + Y_Offset, Velo); 

    // Obsługa pozostałych wycięć
    4, 5, 6, 7, 8:
        sx := _ShapeStart[_CurrentShapeIndex].X;
        sy := _ShapeStart[_CurrentShapeIndex].Y;
        r_val := 10.0;

        IF _CurrentShapeIndex = 4 THEN
            dx := RailSlot;
            dy := ExtrusionLengthY;
        ELSIF _CurrentShapeIndex = 5 THEN
            dx := RailSlot;
            dy := ExtrusionLengthX; 
        ELSIF _CurrentShapeIndex = 6 THEN
            dx := SmallSlot;
            dy := SmallSlot;
        ELSIF _CurrentShapeIndex = 7 THEN
            dx := BigSlot;
            dy := BigSlot;
        ELSIF _CurrentShapeIndex = 8 THEN
            dx := BigSlot;
            dy := BigSlot;
        END_IF

        _GeometryWriter.AddStartPoint(sx, sy);

        _GeometryWriter.AddLine(sx, sy + dy - r_val, Velo);
        IF r_val > 0 THEN
            _GeometryWriter.AddArc(sx + r_val, sy + dy, sx + r_val, sy + dy - r_val, Velo, TRUE);
        END_IF

        _GeometryWriter.AddLine(sx + dx - r_val, sy + dy, Velo);
        IF r_val > 0 THEN
            _GeometryWriter.AddArc(sx + dx, sy + dy - r_val, sx + dx - r_val, sy + dy - r_val, Velo, TRUE);
        END_IF

        _GeometryWriter.AddLine(sx + dx, sy + r_val, Velo);
        IF r_val > 0 THEN
            _GeometryWriter.AddArc(sx + dx - r_val, sy, sx + dx - r_val, sy + r_val, Velo, TRUE);
        END_IF

        _GeometryWriter.AddLine(sx + r_val, sy, Velo);
        IF r_val > 0 THEN
            _GeometryWriter.AddArc(sx, sy + r_val, sx + r_val, sy + r_val, Velo, TRUE);
        END_IF

END_CASE

_GeometryWriter.EndTable();

_Busy := FALSE;
_Done := TRUE;
Build := TRUE;
END_METHOD

METHOD PROTECTED CalculateFootprint
VAR_INPUT
END_VAR
_NominalX := 1200;
_NominalY := 2400;
END_METHOD

PROPERTY ExecutionRoute : E_ExecutionRoute
GET
ExecutionRoute := E_ExecutionRoute.eFeedTable;
END_GET
END_PROPERTY

METHOD FB_init : BOOL
VAR_INPUT
	bInitRetains : BOOL; // if TRUE, the retain variables are initialized (warm start / cold start)
	bInCopyCode : BOOL;  // if TRUE, the instance afterwards gets moved into the copy code (online change)
END_VAR
_Limits.PanelFrontLength.MinVal := 100.0;
_Limits.PanelFrontLength.MaxVal := 2400.0;

_Limits.PanelFrontWidth.MinVal  := 100.0;
_Limits.PanelFrontWidth.MaxVal  := 1200.0;

_Limits.PanelHeight.MinVal      := 0.0;
_Limits.PanelHeight.MaxVal      := 0.0;

_Limits.RailHeightCorrection.MinVal := 0.0;
_Limits.RailHeightCorrection.MaxVal := 0.0;

_Limits.CuttingOverpass.MinVal := 0.0;
_Limits.CuttingOverpass.MaxVal := 50.0;

_Limits.GroovingOverpass.MinVal := 0.0;
_Limits.GroovingOverpass.MaxVal := 50.0;

_Limits.GrooveDepthZ.MinVal := 0.0;
_Limits.GrooveDepthZ.MaxVal := 9.0; 

_Limits.CuttingOverpass.MinVal := 0.0;
_Limits.CuttingOverpass.MaxVal := 50.0;
_Limits.GroovingOverpass.MinVal := 0.0;
_Limits.GroovingOverpass.MaxVal := 50.0;

_Limits.Radius.MinVal := 10.0;     
_Limits.Radius.MaxVal := 600.0;
END_METHOD

END_FUNCTION_BLOCK

// ---- POUs/Builder/Recipes/FB_FeedMeina2_1000x1000.TcPOU
FUNCTION_BLOCK FB_FeedMeina2_1000x1000 EXTENDS FB_RecipeBase

METHOD Build : BOOL
VAR
    TotalX, TotalY, Radius : LREAL;
    Velo : LREAL;
    localConfig : ST_GantryXYZ_Config;
	
    // Zmienne do otworów
    HoleDistanceFromEdgeOfRail : LREAL := 100.0;
    SomeFixedDimension         : LREAL := 12.63;
    PanelRailOffsetX           : LREAL;
    PanelRailOffsetY           : LREAL;
    ExtrusionLengthX           : LREAL;
    ExtrusionLengthY           : LREAL;
    
    NumberOfHolesX             : INT := 3;
    NumberOfHolesY             : INT := 5;
    HolesSpacingX              : LREAL;
    HolesSpacingY              : LREAL;
    
    i                          : INT;
    holeIdx                    : INT;
	
	RailSlot  : LREAL := 29.0;
	BigSlot   : LREAL := 200.0;
	SmallSlot : LREAL := 100.0;

// Zmienne pomocnicze do generowania ścieżek
	sx : LREAL;
	sy : LREAL;
	dx : LREAL;
	dy : LREAL;
	r_val : LREAL;
	
	PanelGap : LREAL := 20.0; 
    Y_Offset : LREAL;
    p        : INT;
	
END_VAR
_Busy := TRUE;
_Done := FALSE;
_Error := FALSE;
Build := FALSE;
THIS^.UpdateNestingLimits();

IF NOT _Config.IsValid THEN
    _Busy := FALSE;
    _Error := TRUE; 
    Build := FALSE;
    RETURN;
END_IF

// ===================================================
// NOWE GEOMETRIE DLA DWÓCH KWADRATÓW (W OSI Y)
// ===================================================
TotalX := 1000.0; 
TotalY := 1000.0; 
Radius := _Config.Radius;

IF Radius > (TotalX / 2.0) THEN Radius := TotalX / 2.0; END_IF
IF Radius > (TotalY / 2.0) THEN Radius := TotalY / 2.0; END_IF

// Przerwa między panelami (20 mm) w osi Y
PanelGap := 20.0; 

// Offsety dla szyn
PanelRailOffsetX := 0.1 * TotalX;
PanelRailOffsetY := 0.1 * TotalY;

ExtrusionLengthX := TotalX - (2.0 * PanelRailOffsetX);
ExtrusionLengthY := TotalY - (2.0 * PanelRailOffsetY);

// Wyliczenie rozstawu otworów
IF NumberOfHolesX > 1 THEN
    HolesSpacingX := (ExtrusionLengthX - (2.0 * HoleDistanceFromEdgeOfRail)) / INT_TO_LREAL(NumberOfHolesX - 1);
ELSE
    HolesSpacingX := 0.0;
END_IF

IF NumberOfHolesY > 1 THEN
    HolesSpacingY := (ExtrusionLengthY - (2.0 * HoleDistanceFromEdgeOfRail)) / INT_TO_LREAL(NumberOfHolesY - 1);
ELSE
    HolesSpacingY := 0.0;
END_IF


// ===================================================
// GENEROWANIE OTWORÓW DLA OBU PANELÓW (OFFSET W Y)
// ===================================================
holeIdx := 0; 

FOR p := 0 TO 1 DO
    // Wyznaczamy offset Y dla aktualnego panelu (Panel 1: 0.0, Panel 2: 1020.0)
    Y_Offset := INT_TO_LREAL(p) * (TotalY + PanelGap);

    // 1. Otwór na dokładnym środku danego panelu
    holeIdx := holeIdx + 1;
    _HolesDrill[holeIdx].X := LREAL_TO_REAL(TotalX / 2.0);
    _HolesDrill[holeIdx].Y := LREAL_TO_REAL((TotalY / 2.0) + Y_Offset);

    // 2. Rail Y1 (Lewa)
    FOR i := NumberOfHolesY TO 1 BY -1 DO
        holeIdx := holeIdx + 1;
        _HolesDrill[holeIdx].X := LREAL_TO_REAL(PanelRailOffsetX - SomeFixedDimension);
        _HolesDrill[holeIdx].Y := LREAL_TO_REAL(PanelRailOffsetY + HoleDistanceFromEdgeOfRail + ((i - 1) * HolesSpacingY) + Y_Offset);
    END_FOR

    // 3. Rail X1 (Dolna)
    FOR i := 1 TO NumberOfHolesX DO
        holeIdx := holeIdx + 1;
        _HolesDrill[holeIdx].X := LREAL_TO_REAL(PanelRailOffsetX + HoleDistanceFromEdgeOfRail + ((i - 1) * HolesSpacingX));
        _HolesDrill[holeIdx].Y := LREAL_TO_REAL(PanelRailOffsetY - SomeFixedDimension + Y_Offset);
    END_FOR

    // 4. Rail Y2 (Prawa)
    FOR i := 1 TO NumberOfHolesY DO
        holeIdx := holeIdx + 1;
        _HolesDrill[holeIdx].X := LREAL_TO_REAL(PanelRailOffsetX + ExtrusionLengthX + SomeFixedDimension);
        _HolesDrill[holeIdx].Y := LREAL_TO_REAL(PanelRailOffsetY + HoleDistanceFromEdgeOfRail + ((i - 1) * HolesSpacingY) + Y_Offset);
    END_FOR

    // 5. Rail X2 (Górna)
    FOR i := NumberOfHolesX TO 1 BY -1 DO
        holeIdx := holeIdx + 1;
        _HolesDrill[holeIdx].X := LREAL_TO_REAL(PanelRailOffsetX + HoleDistanceFromEdgeOfRail + ((i - 1) * HolesSpacingX));
        _HolesDrill[holeIdx].Y := LREAL_TO_REAL(PanelRailOffsetY + ExtrusionLengthY + SomeFixedDimension + Y_Offset);
    END_FOR
END_FOR

_HolesToDrill := holeIdx;

// ===================================================
// DEFINICJA ILOŚCI I PUNKTÓW STARTOWYCH (Dla FeedTable)
// ===================================================
_ShapesCount := 7; 

// 1. Kształt główny - Panel Dolny
_ShapeStart[1].X := 0.0;
_ShapeStart[1].Y := 0.0;

// 2. Kształt główny - Panel Górny (Wysokość 1000 + 20 przerwy w osi Y)
_ShapeStart[2].X := 0.0;
_ShapeStart[2].Y := TotalY + PanelGap; // Czyli 1020.0

// Pozostałe kształty bez zmian (są powyżej 2150 w Y, więc nie kolidują z kwadratami)
_ShapeStart[3].X := 1030.0;
_ShapeStart[3].Y := 0.0;

_ShapeStart[4].X := 1090.0;
_ShapeStart[4].Y := 0.0;

_ShapeStart[5].X := 210.0;
_ShapeStart[5].Y := 2200.0;

_ShapeStart[6].X := 410.0;
_ShapeStart[6].Y := 2150.0;

_ShapeStart[7].X := 810.0;
_ShapeStart[7].Y := 2150.0;


IF _ConfigProvider <> 0 THEN
    localConfig := _ConfigProvider.Config;
    Velo := localConfig.CuttingSpeedXY;
ELSE
    Velo := 50.0;
END_IF

_GeometryWriter.Clear();
_GeometryWriter.EnableTangentialFollowing();

sx := 0.0; sy := 0.0; dx := 0.0; dy := 0.0; r_val := 0.0;

// RYSOWANIE KSZTAŁTU ZGODNIE Z INDEKSEM
CASE _CurrentShapeIndex OF
    1, 2:
        sx := _ShapeStart[_CurrentShapeIndex].X;
        sy := _ShapeStart[_CurrentShapeIndex].Y;

        _GeometryWriter.AddStartPoint(sx, sy);

        _GeometryWriter.AddLine(sx, sy + TotalY - Radius, Velo);
        IF Radius > 0 THEN
            _GeometryWriter.AddArc(sx + Radius, sy + TotalY, sx + Radius, sy + TotalY - Radius, Velo, TRUE);
        END_IF

        _GeometryWriter.AddLine(sx + TotalX - Radius, sy + TotalY, Velo);
        IF Radius > 0 THEN
            _GeometryWriter.AddArc(sx + TotalX, sy + TotalY - Radius, sx + TotalX - Radius, sy + TotalY - Radius, Velo, TRUE);
        END_IF

        _GeometryWriter.AddLine(sx + TotalX, sy + Radius, Velo);
        IF Radius > 0 THEN
            _GeometryWriter.AddArc(sx + TotalX - Radius, sy, sx + TotalX - Radius, sy + Radius, Velo, TRUE);
        END_IF

        _GeometryWriter.AddLine(sx + Radius, sy, Velo);
        IF Radius > 0 THEN
            _GeometryWriter.AddArc(sx, sy + Radius, sx + Radius, sy + Radius, Velo, TRUE);
        END_IF

    3, 4, 5, 6, 7:
        sx := _ShapeStart[_CurrentShapeIndex].X;
        sy := _ShapeStart[_CurrentShapeIndex].Y;
        r_val := 10.0;

        IF _CurrentShapeIndex = 3 THEN
            dx := RailSlot;
            dy := ExtrusionLengthY;
        ELSIF _CurrentShapeIndex = 4 THEN
            dx := RailSlot;
            dy := ExtrusionLengthX; 
        ELSIF _CurrentShapeIndex = 5 THEN
            dx := SmallSlot;
            dy := SmallSlot;
        ELSIF _CurrentShapeIndex = 6 THEN
            dx := BigSlot;
            dy := BigSlot;
        ELSIF _CurrentShapeIndex = 7 THEN
            dx := BigSlot;
            dy := BigSlot;
        END_IF

        _GeometryWriter.AddStartPoint(sx, sy);

        _GeometryWriter.AddLine(sx, sy + dy - r_val, Velo);
        IF r_val > 0 THEN
            _GeometryWriter.AddArc(sx + r_val, sy + dy, sx + r_val, sy + dy - r_val, Velo, TRUE);
        END_IF

        _GeometryWriter.AddLine(sx + dx - r_val, sy + dy, Velo);
        IF r_val > 0 THEN
            _GeometryWriter.AddArc(sx + dx, sy + dy - r_val, sx + dx - r_val, sy + dy - r_val, Velo, TRUE);
        END_IF

        _GeometryWriter.AddLine(sx + dx, sy + r_val, Velo);
        IF r_val > 0 THEN
            _GeometryWriter.AddArc(sx + dx - r_val, sy, sx + dx - r_val, sy + r_val, Velo, TRUE);
        END_IF

        _GeometryWriter.AddLine(sx + r_val, sy, Velo);
        IF r_val > 0 THEN
            _GeometryWriter.AddArc(sx, sy + r_val, sx + r_val, sy + r_val, Velo, TRUE);
        END_IF

END_CASE

_GeometryWriter.EndTable();

_Busy := FALSE;
_Done := TRUE;
Build := TRUE;
END_METHOD

METHOD PROTECTED CalculateFootprint
VAR_INPUT
END_VAR
_NominalX := 1200;
_NominalY := 2400;
END_METHOD

PROPERTY ExecutionRoute : E_ExecutionRoute
GET
ExecutionRoute := E_ExecutionRoute.eFeedTable;
END_GET
END_PROPERTY

METHOD FB_init : BOOL
VAR_INPUT
	bInitRetains : BOOL; // if TRUE, the retain variables are initialized (warm start / cold start)
	bInCopyCode : BOOL;  // if TRUE, the instance afterwards gets moved into the copy code (online change)
END_VAR
_Limits.PanelFrontLength.MinVal := 100.0;
_Limits.PanelFrontLength.MaxVal := 2400.0;

_Limits.PanelFrontWidth.MinVal  := 100.0;
_Limits.PanelFrontWidth.MaxVal  := 1200.0;

_Limits.PanelHeight.MinVal      := 0.0;
_Limits.PanelHeight.MaxVal      := 0.0;

_Limits.RailHeightCorrection.MinVal := 0.0;
_Limits.RailHeightCorrection.MaxVal := 0.0;

_Limits.CuttingOverpass.MinVal := 0.0;
_Limits.CuttingOverpass.MaxVal := 50.0;

_Limits.GroovingOverpass.MinVal := 0.0;
_Limits.GroovingOverpass.MaxVal := 50.0;

_Limits.GrooveDepthZ.MinVal := 0.0;
_Limits.GrooveDepthZ.MaxVal := 9.0; 

_Limits.CuttingOverpass.MinVal := 0.0;
_Limits.CuttingOverpass.MaxVal := 50.0;
_Limits.GroovingOverpass.MinVal := 0.0;
_Limits.GroovingOverpass.MaxVal := 50.0;

_Limits.Radius.MinVal := 10.0;     
_Limits.Radius.MaxVal := 600.0;
END_METHOD

END_FUNCTION_BLOCK

// ---- POUs/Builder/Recipes/FB_FeedMeina2_1000x1000_Circles.TcPOU
FUNCTION_BLOCK FB_FeedMeina2_1000x1000_Circles EXTENDS FB_RecipeBase

METHOD Build : BOOL
VAR
    TotalX, TotalY, Radius : LREAL;
    CircleRadius           : LREAL;
    Velo                   : LREAL;
    localConfig            : ST_GantryXYZ_Config;
    
    PanelGap               : LREAL;
    Y_Offset               : LREAL;
    p                      : INT;

    HoleDistanceFromEdgeOfRail : LREAL := 100.0;
    SomeFixedDimension         : LREAL := 12.63;
    PanelRailOffsetX           : LREAL;
    PanelRailOffsetY           : LREAL;
    ExtrusionLengthX           : LREAL;
    ExtrusionLengthY           : LREAL;
    
    NumberOfHolesX             : INT := 3;
    NumberOfHolesY             : INT := 5;
    HolesSpacingX              : LREAL;
    HolesSpacingY              : LREAL;
    
    i                          : INT;
    holeIdx                    : INT;
    
    RailSlot  : LREAL := 29.0;
    BigSlot   : LREAL := 200.0;
    SmallSlot : LREAL := 100.0;

    LeadInY   : LREAL := 10.0;
    LeadOutY  : LREAL := 10.0;

    sx : LREAL;
    sy : LREAL;
    dx : LREAL;
    dy : LREAL;
    r_val : LREAL;
END_VAR
_Busy := TRUE;
_Done := FALSE;
_Error := FALSE;
Build := FALSE;
THIS^.UpdateNestingLimits();

IF NOT _Config.IsValid THEN
    _Busy := FALSE;
    _Error := TRUE; 
    Build := FALSE;
    RETURN;
END_IF

TotalX := 1000.0;
TotalY := 1000.0;
CircleRadius := TotalX / 2.0;

PanelGap := 20.0; 

PanelRailOffsetX := 0.1 * TotalX;
PanelRailOffsetY := 0.1 * TotalY;

ExtrusionLengthX := TotalX - (2.0 * PanelRailOffsetX);
ExtrusionLengthY := TotalY - (2.0 * PanelRailOffsetY);

IF NumberOfHolesX > 1 THEN
    HolesSpacingX := (ExtrusionLengthX - (2.0 * HoleDistanceFromEdgeOfRail)) / INT_TO_LREAL(NumberOfHolesX - 1);
ELSE
    HolesSpacingX := 0.0;
END_IF

IF NumberOfHolesY > 1 THEN
    HolesSpacingY := (ExtrusionLengthY - (2.0 * HoleDistanceFromEdgeOfRail)) / INT_TO_LREAL(NumberOfHolesY - 1);
ELSE
    HolesSpacingY := 0.0;
END_IF

holeIdx := 0; 

FOR p := 0 TO 1 DO
    Y_Offset := INT_TO_LREAL(p) * (TotalY + PanelGap);

    holeIdx := holeIdx + 1;
    _HolesDrill[holeIdx].X := LREAL_TO_REAL(TotalX / 2.0);
    _HolesDrill[holeIdx].Y := LREAL_TO_REAL((TotalY / 2.0) + Y_Offset);

    FOR i := NumberOfHolesY TO 1 BY -1 DO
        holeIdx := holeIdx + 1;
        _HolesDrill[holeIdx].X := LREAL_TO_REAL(PanelRailOffsetX - SomeFixedDimension);
        _HolesDrill[holeIdx].Y := LREAL_TO_REAL(PanelRailOffsetY + HoleDistanceFromEdgeOfRail + ((i - 1) * HolesSpacingY) + Y_Offset);
    END_FOR

    FOR i := 1 TO NumberOfHolesX DO
        holeIdx := holeIdx + 1;
        _HolesDrill[holeIdx].X := LREAL_TO_REAL(PanelRailOffsetX + HoleDistanceFromEdgeOfRail + ((i - 1) * HolesSpacingX));
        _HolesDrill[holeIdx].Y := LREAL_TO_REAL(PanelRailOffsetY - SomeFixedDimension + Y_Offset);
    END_FOR

    FOR i := 1 TO NumberOfHolesY DO
        holeIdx := holeIdx + 1;
        _HolesDrill[holeIdx].X := LREAL_TO_REAL(PanelRailOffsetX + ExtrusionLengthX + SomeFixedDimension);
        _HolesDrill[holeIdx].Y := LREAL_TO_REAL(PanelRailOffsetY + HoleDistanceFromEdgeOfRail + ((i - 1) * HolesSpacingY) + Y_Offset);
    END_FOR

    FOR i := NumberOfHolesX TO 1 BY -1 DO
        holeIdx := holeIdx + 1;
        _HolesDrill[holeIdx].X := LREAL_TO_REAL(PanelRailOffsetX + HoleDistanceFromEdgeOfRail + ((i - 1) * HolesSpacingX));
        _HolesDrill[holeIdx].Y := LREAL_TO_REAL(PanelRailOffsetY + ExtrusionLengthY + SomeFixedDimension + Y_Offset);
    END_FOR
END_FOR

_HolesToDrill := holeIdx;

_ShapesCount := 7; 

_ShapeStart[1].X := TotalX;
_ShapeStart[1].Y := CircleRadius - LeadInY;

_ShapeStart[2].X := TotalX;
_ShapeStart[2].Y := TotalY + PanelGap + CircleRadius - LeadInY;

_ShapeStart[3].X := 1030.0;
_ShapeStart[3].Y := 0.0;

_ShapeStart[4].X := 1090.0;
_ShapeStart[4].Y := 0.0;

_ShapeStart[5].X := 210.0;
_ShapeStart[5].Y := 2200.0;

_ShapeStart[6].X := 410.0;
_ShapeStart[6].Y := 2150.0;

_ShapeStart[7].X := 810.0;
_ShapeStart[7].Y := 2150.0;

IF _ConfigProvider <> 0 THEN
    localConfig := _ConfigProvider.Config;
    Velo := localConfig.CuttingSpeedXY;
ELSE
    Velo := 50.0;
END_IF

_GeometryWriter.Clear();
_GeometryWriter.EnableTangentialFollowing();

sx := 0.0; sy := 0.0; dx := 0.0; dy := 0.0; r_val := 0.0;

CASE _CurrentShapeIndex OF
    1, 2:
        IF _CurrentShapeIndex = 1 THEN
            Y_Offset := 0.0;
        ELSE
            Y_Offset := TotalY + PanelGap;
        END_IF

        _GeometryWriter.AddStartPoint(_ShapeStart[_CurrentShapeIndex].X, _ShapeStart[_CurrentShapeIndex].Y); 
        _GeometryWriter.AddLine(TotalX, CircleRadius + Y_Offset, Velo); 
        _GeometryWriter.AddArc(0.0, CircleRadius + Y_Offset, CircleRadius, CircleRadius + Y_Offset, Velo, FALSE);
        _GeometryWriter.AddArc(TotalX, CircleRadius + Y_Offset, CircleRadius, CircleRadius + Y_Offset, Velo, FALSE);
        _GeometryWriter.AddLine(TotalX, CircleRadius + LeadOutY + Y_Offset, Velo); 

    3, 4, 5, 6, 7:
        sx := _ShapeStart[_CurrentShapeIndex].X;
        sy := _ShapeStart[_CurrentShapeIndex].Y;
        r_val := 10.0;

        IF _CurrentShapeIndex = 3 THEN
            dx := RailSlot;
            dy := ExtrusionLengthY;
        ELSIF _CurrentShapeIndex = 4 THEN
            dx := RailSlot;
            dy := ExtrusionLengthX; 
        ELSIF _CurrentShapeIndex = 5 THEN
            dx := SmallSlot;
            dy := SmallSlot;
        ELSIF _CurrentShapeIndex = 6 THEN
            dx := BigSlot;
            dy := BigSlot;
        ELSIF _CurrentShapeIndex = 7 THEN
            dx := BigSlot;
            dy := BigSlot;
        END_IF

        _GeometryWriter.AddStartPoint(sx, sy);

        _GeometryWriter.AddLine(sx, sy + dy - r_val, Velo);
        IF r_val > 0 THEN
            _GeometryWriter.AddArc(sx + r_val, sy + dy, sx + r_val, sy + dy - r_val, Velo, TRUE);
        END_IF

        _GeometryWriter.AddLine(sx + dx - r_val, sy + dy, Velo);
        IF r_val > 0 THEN
            _GeometryWriter.AddArc(sx + dx, sy + dy - r_val, sx + dx - r_val, sy + dy - r_val, Velo, TRUE);
        END_IF

        _GeometryWriter.AddLine(sx + dx, sy + r_val, Velo);
        IF r_val > 0 THEN
            _GeometryWriter.AddArc(sx + dx - r_val, sy, sx + dx - r_val, sy + r_val, Velo, TRUE);
        END_IF

        _GeometryWriter.AddLine(sx + r_val, sy, Velo);
        IF r_val > 0 THEN
            _GeometryWriter.AddArc(sx, sy + r_val, sx + r_val, sy + r_val, Velo, TRUE);
        END_IF

END_CASE

_GeometryWriter.EndTable();

_Busy := FALSE;
_Done := TRUE;
Build := TRUE;
END_METHOD

METHOD PROTECTED CalculateFootprint
VAR_INPUT
END_VAR
_NominalX := 1200;
_NominalY := 2400;
END_METHOD

PROPERTY ExecutionRoute : E_ExecutionRoute
GET
ExecutionRoute := E_ExecutionRoute.eFeedTable;
END_GET
END_PROPERTY

METHOD FB_init : BOOL
VAR_INPUT
	bInitRetains : BOOL; // if TRUE, the retain variables are initialized (warm start / cold start)
	bInCopyCode : BOOL;  // if TRUE, the instance afterwards gets moved into the copy code (online change)
END_VAR
_Limits.PanelFrontLength.MinVal := 100.0;
_Limits.PanelFrontLength.MaxVal := 2400.0;

_Limits.PanelFrontWidth.MinVal  := 100.0;
_Limits.PanelFrontWidth.MaxVal  := 1200.0;

_Limits.PanelHeight.MinVal      := 0.0;
_Limits.PanelHeight.MaxVal      := 0.0;

_Limits.RailHeightCorrection.MinVal := 0.0;
_Limits.RailHeightCorrection.MaxVal := 0.0;

_Limits.CuttingOverpass.MinVal := 0.0;
_Limits.CuttingOverpass.MaxVal := 50.0;

_Limits.GroovingOverpass.MinVal := 0.0;
_Limits.GroovingOverpass.MaxVal := 50.0;

_Limits.GrooveDepthZ.MinVal := 0.0;
_Limits.GrooveDepthZ.MaxVal := 9.0; 

_Limits.CuttingOverpass.MinVal := 0.0;
_Limits.CuttingOverpass.MaxVal := 50.0;
_Limits.GroovingOverpass.MinVal := 0.0;
_Limits.GroovingOverpass.MaxVal := 50.0;

_Limits.Radius.MinVal := 10.0;     
_Limits.Radius.MaxVal := 600.0;
END_METHOD

END_FUNCTION_BLOCK

// ---- POUs/Builder/Recipes/FB_FeedMeina2_2000x500.TcPOU
FUNCTION_BLOCK FB_FeedMeina2_2000x500 EXTENDS FB_RecipeBase

METHOD Build : BOOL
VAR
    TotalX, TotalY, Radius : LREAL;
    Velo : LREAL;
    localConfig : ST_GantryXYZ_Config;
	
    // Zmienne do otworów
    HoleDistanceFromEdgeOfRail : LREAL := 100.0;
    SomeFixedDimension         : LREAL := 12.63;
    PanelRailOffsetX           : LREAL;
    PanelRailOffsetY           : LREAL;
    ExtrusionLengthX           : LREAL;
    ExtrusionLengthY           : LREAL;
    
    NumberOfHolesX             : INT := 3;
    NumberOfHolesY             : INT := 5;
    HolesSpacingX              : LREAL;
    HolesSpacingY              : LREAL;
    
    i                          : INT;
    holeIdx                    : INT;
	
	RailSlot  : LREAL := 29.0;
	BigSlot   : LREAL := 200.0;
	SmallSlot : LREAL := 100.0;

// Zmienne pomocnicze do generowania ścieżek
	sx : LREAL;
	sy : LREAL;
	dx : LREAL;
	dy : LREAL;
	r_val : LREAL;
	
	PanelGap : LREAL := 20.0; 
    X_Offset : LREAL;
    p        : INT;
	
END_VAR
_Busy := TRUE;
_Done := FALSE;
_Error := FALSE;
Build := FALSE;
THIS^.UpdateNestingLimits();

IF NOT _Config.IsValid THEN
    _Busy := FALSE;
    _Error := TRUE; 
    Build := FALSE;
    RETURN;
END_IF

// ===================================================
// NOWE GEOMETRIE DLA DWÓCH PANELÓW
// ===================================================
// Pojedynczy panel ma teraz szerokość 500 mm, a długość 2000 mm
TotalX := 500.0; 
TotalY := 2000.0; 
Radius := _Config.Radius;

IF Radius > (TotalX / 2.0) THEN Radius := TotalX / 2.0; END_IF
IF Radius > (TotalY / 2.0) THEN Radius := TotalY / 2.0; END_IF

// Przerwa między panelami (2 cm = 20 mm)
PanelGap := 20.0; 

// Offsety dla szyn (zachowujemy oryginalne proporcje 10% wymiaru gabarytowego)
PanelRailOffsetX := 0.1 * TotalX;
PanelRailOffsetY := 0.1 * TotalY;

ExtrusionLengthX := TotalX - (2.0 * PanelRailOffsetX);
ExtrusionLengthY := TotalY - (2.0 * PanelRailOffsetY);

// Wyliczenie rozstawu otworów (dla pojedynczego panelu)
IF NumberOfHolesX > 1 THEN
    HolesSpacingX := (ExtrusionLengthX - (2.0 * HoleDistanceFromEdgeOfRail)) / INT_TO_LREAL(NumberOfHolesX - 1);
ELSE
    HolesSpacingX := 0.0;
END_IF

IF NumberOfHolesY > 1 THEN
    HolesSpacingY := (ExtrusionLengthY - (2.0 * HoleDistanceFromEdgeOfRail)) / INT_TO_LREAL(NumberOfHolesY - 1);
ELSE
    HolesSpacingY := 0.0;
END_IF


// ===================================================
// GENEROWANIE OTWORÓW DLA OBU PANELÓW
// ===================================================
holeIdx := 0; // Startujemy od 0, indeks zwiększany wewnątrz

// Pętla po dwóch panelach (p = 0 dla pierwszego, p = 1 dla drugiego)
FOR p := 0 TO 1 DO
    // Wyznaczamy offset X dla aktualnego panelu (Panel 1: 0.0, Panel 2: 520.0)
    X_Offset := INT_TO_LREAL(p) * (TotalX + PanelGap);

    // 1. Otwór na dokładnym środku danego panelu
    holeIdx := holeIdx + 1;
    _HolesDrill[holeIdx].X := LREAL_TO_REAL((TotalX / 2.0) + X_Offset);
    _HolesDrill[holeIdx].Y := LREAL_TO_REAL(TotalY / 2.0);

    // 2. Rail Y1 (Lewa)
    FOR i := NumberOfHolesY TO 1 BY -1 DO
        holeIdx := holeIdx + 1;
        _HolesDrill[holeIdx].X := LREAL_TO_REAL(PanelRailOffsetX - SomeFixedDimension + X_Offset);
        _HolesDrill[holeIdx].Y := LREAL_TO_REAL(PanelRailOffsetY + HoleDistanceFromEdgeOfRail + ((i - 1) * HolesSpacingY));
    END_FOR

    // 3. Rail X1 (Dolna)
    FOR i := 1 TO NumberOfHolesX DO
        holeIdx := holeIdx + 1;
        _HolesDrill[holeIdx].X := LREAL_TO_REAL(PanelRailOffsetX + HoleDistanceFromEdgeOfRail + ((i - 1) * HolesSpacingX) + X_Offset);
        _HolesDrill[holeIdx].Y := LREAL_TO_REAL(PanelRailOffsetY - SomeFixedDimension);
    END_FOR

    // 4. Rail Y2 (Prawa)
    FOR i := 1 TO NumberOfHolesY DO
        holeIdx := holeIdx + 1;
        _HolesDrill[holeIdx].X := LREAL_TO_REAL(PanelRailOffsetX + ExtrusionLengthX + SomeFixedDimension + X_Offset);
        _HolesDrill[holeIdx].Y := LREAL_TO_REAL(PanelRailOffsetY + HoleDistanceFromEdgeOfRail + ((i - 1) * HolesSpacingY));
    END_FOR

    // 5. Rail X2 (Górna)
    FOR i := NumberOfHolesX TO 1 BY -1 DO
        holeIdx := holeIdx + 1;
        _HolesDrill[holeIdx].X := LREAL_TO_REAL(PanelRailOffsetX + HoleDistanceFromEdgeOfRail + ((i - 1) * HolesSpacingX) + X_Offset);
        _HolesDrill[holeIdx].Y := LREAL_TO_REAL(PanelRailOffsetY + ExtrusionLengthY + SomeFixedDimension);
    END_FOR
END_FOR

// Przypisanie całkowitej liczby otworów z obu paneli
_HolesToDrill := holeIdx;


// ===================================================
// DEFINICJA ILOŚCI I PUNKTÓW STARTOWYCH (Dla FeedTable)
// ===================================================
_ShapesCount := 7; // ZWIĘKSZONO O 1: Teraz mamy 2 główne panele + 5 wycięć z tabeli

// 1. Kształt główny - Panel Lewy
_ShapeStart[1].X := 0.0;
_ShapeStart[1].Y := 0.0;

// 2. Kształt główny - Panel Prawy (szerokość 500 + 20 przerwy)
_ShapeStart[2].X := TotalX + PanelGap; // Czyli 520.0
_ShapeStart[2].Y := 0.0;

// Przesunięcie pozostałych kształtów z tabeli o jeden indeks w górę (były 2..6, są 3..7)
// 3. No. 1
_ShapeStart[3].X := 1030.0;
_ShapeStart[3].Y := 0.0;

// 4. No. 2
_ShapeStart[4].X := 1090.0;
_ShapeStart[4].Y := 0.0;

// 5. No. 3
_ShapeStart[5].X := 210.0;
_ShapeStart[5].Y := 2200.0;

// 6. No. 4
_ShapeStart[6].X := 410.0;
_ShapeStart[6].Y := 2150.0;

// 7. No. 5
_ShapeStart[7].X := 810.0;
_ShapeStart[7].Y := 2150.0;


IF _ConfigProvider <> 0 THEN
    localConfig := _ConfigProvider.Config;
    Velo := localConfig.CuttingSpeedXY;
ELSE
    Velo := 50.0;
END_IF

_GeometryWriter.Clear();
_GeometryWriter.EnableTangentialFollowing();

// Reset zmiennych pomocniczych
sx := 0.0; sy := 0.0; dx := 0.0; dy := 0.0; r_val := 0.0;

// RYSOWANIE KSZTAŁTU ZGODNIE Z INDEKSEM
CASE _CurrentShapeIndex OF
    1, 2:
        // ==========================================
        // KSZTAŁT 1 i 2 (Dwa identyczne panele główne)
        // ==========================================
        // Pobieramy punkt startowy odpowiedni dla Panelu 1 (0,0) lub Panelu 2 (520,0)
        sx := _ShapeStart[_CurrentShapeIndex].X;
        sy := _ShapeStart[_CurrentShapeIndex].Y;

        _GeometryWriter.AddStartPoint(sx, sy);

        // Krawędzie rysowane są z uwzględnieniem punktu startowego 'sx' oraz 'sy'
        _GeometryWriter.AddLine(sx, sy + TotalY - Radius, Velo);
        IF Radius > 0 THEN
            _GeometryWriter.AddArc(sx + Radius, sy + TotalY, sx + Radius, sy + TotalY - Radius, Velo, TRUE);
        END_IF

        _GeometryWriter.AddLine(sx + TotalX - Radius, sy + TotalY, Velo);
        IF Radius > 0 THEN
            _GeometryWriter.AddArc(sx + TotalX, sy + TotalY - Radius, sx + TotalX - Radius, sy + TotalY - Radius, Velo, TRUE);
        END_IF

        _GeometryWriter.AddLine(sx + TotalX, sy + Radius, Velo);
        IF Radius > 0 THEN
            _GeometryWriter.AddArc(sx + TotalX - Radius, sy, sx + TotalX - Radius, sy + Radius, Velo, TRUE);
        END_IF

        _GeometryWriter.AddLine(sx + Radius, sy, Velo);
        IF Radius > 0 THEN
            _GeometryWriter.AddArc(sx, sy + Radius, sx + Radius, sy + Radius, Velo, TRUE);
        END_IF

    3, 4, 5, 6, 7:
        // ==========================================
        // KSZTAŁTY OD 3 DO 7 (Dawne 2 do 6)
        // ==========================================
        sx := _ShapeStart[_CurrentShapeIndex].X;
        sy := _ShapeStart[_CurrentShapeIndex].Y;
        r_val := 10.0;

        // Dopasowanie indeksów warunków (zmniejszone o 1 w stosunku do _CurrentShapeIndex)
        IF _CurrentShapeIndex = 3 THEN
            dx := RailSlot;
            dy := ExtrusionLengthY;
        ELSIF _CurrentShapeIndex = 4 THEN
            dx := RailSlot;
            dy := ExtrusionLengthX; // Uwaga: ExtrusionLengthX bazuje teraz na nowym TotalX (500)
        ELSIF _CurrentShapeIndex = 5 THEN
            dx := SmallSlot;
            dy := SmallSlot;
        ELSIF _CurrentShapeIndex = 6 THEN
            dx := BigSlot;
            dy := BigSlot;
        ELSIF _CurrentShapeIndex = 7 THEN
            dx := BigSlot;
            dy := BigSlot;
        END_IF

        _GeometryWriter.AddStartPoint(sx, sy);

        // 1. Lewa krawędź w górę
        _GeometryWriter.AddLine(sx, sy + dy - r_val, Velo);
        IF r_val > 0 THEN
            _GeometryWriter.AddArc(sx + r_val, sy + dy, sx + r_val, sy + dy - r_val, Velo, TRUE);
        END_IF

        // 2. Górna krawędź w prawo
        _GeometryWriter.AddLine(sx + dx - r_val, sy + dy, Velo);
        IF r_val > 0 THEN
            _GeometryWriter.AddArc(sx + dx, sy + dy - r_val, sx + dx - r_val, sy + dy - r_val, Velo, TRUE);
        END_IF

        // 3. Prawa krawędź w dół
        _GeometryWriter.AddLine(sx + dx, sy + r_val, Velo);
        IF r_val > 0 THEN
            _GeometryWriter.AddArc(sx + dx - r_val, sy, sx + dx - r_val, sy + r_val, Velo, TRUE);
        END_IF

        // 4. Dolna krawędź w lewo i zamknięcie
        _GeometryWriter.AddLine(sx + r_val, sy, Velo);
        IF r_val > 0 THEN
            _GeometryWriter.AddArc(sx, sy + r_val, sx + r_val, sy + r_val, Velo, TRUE);
        END_IF

END_CASE

_GeometryWriter.EndTable();

_Busy := FALSE;
_Done := TRUE;
Build := TRUE;
END_METHOD

METHOD PROTECTED CalculateFootprint
VAR_INPUT
END_VAR
_NominalX := 1200;
_NominalY := 2400;
END_METHOD

PROPERTY ExecutionRoute : E_ExecutionRoute
GET
ExecutionRoute := E_ExecutionRoute.eFeedTable;
END_GET
END_PROPERTY

METHOD FB_init : BOOL
VAR_INPUT
	bInitRetains : BOOL; // if TRUE, the retain variables are initialized (warm start / cold start)
	bInCopyCode : BOOL;  // if TRUE, the instance afterwards gets moved into the copy code (online change)
END_VAR
_Limits.PanelFrontLength.MinVal := 100.0;
_Limits.PanelFrontLength.MaxVal := 2400.0;

_Limits.PanelFrontWidth.MinVal  := 100.0;
_Limits.PanelFrontWidth.MaxVal  := 1200.0;

_Limits.PanelHeight.MinVal      := 0.0;
_Limits.PanelHeight.MaxVal      := 0.0;

_Limits.RailHeightCorrection.MinVal := 0.0;
_Limits.RailHeightCorrection.MaxVal := 0.0;

_Limits.CuttingOverpass.MinVal := 0.0;
_Limits.CuttingOverpass.MaxVal := 50.0;

_Limits.GroovingOverpass.MinVal := 0.0;
_Limits.GroovingOverpass.MaxVal := 50.0;

_Limits.GrooveDepthZ.MinVal := 0.0;
_Limits.GrooveDepthZ.MaxVal := 9.0; 

_Limits.CuttingOverpass.MinVal := 0.0;
_Limits.CuttingOverpass.MaxVal := 50.0;
_Limits.GroovingOverpass.MinVal := 0.0;
_Limits.GroovingOverpass.MaxVal := 50.0;

_Limits.Radius.MinVal := 10.0;     
_Limits.Radius.MaxVal := 600.0;
END_METHOD

END_FUNCTION_BLOCK

// ---- POUs/Builder/Recipes/FB_FeedMeina2_Samples.TcPOU
FUNCTION_BLOCK FB_FeedMeina2_Samples EXTENDS FB_RecipeBase

METHOD Build : BOOL
VAR
    TotalX : REAL;
    TotalY : REAL;
    Radius : REAL;
    Velo   : REAL;
    localConfig : ST_GantryXYZ_Config;

    PanelRailOffsetX : REAL;
    PanelRailOffsetY : REAL;
    ExtrusionLengthX : REAL;
    ExtrusionLengthY : REAL;
    
    NumberOfHolesX : INT := 2; 
    NumberOfHolesY : INT := 2;
    HoleDistanceFromEdgeOfRail : REAL := 25.0;
    SomeFixedDimension : REAL := 12.63; 
    
    HolesSpacingX : LREAL;
    HolesSpacingY : LREAL;
    
    holeIdx : INT;
    i       : INT;
END_VAR
_Busy := TRUE;
_Done := FALSE;
_Error := FALSE;
Build := FALSE;
THIS^.UpdateNestingLimits();

IF NOT _Config.IsValid THEN
    _Busy := FALSE;
    _Error := TRUE; 
    Build := FALSE;
    RETURN;
END_IF

// ===================================================
// GABARYTY I PRĘDKOŚĆ
// ===================================================
TotalX := _Config.PanelFrontWidth;
TotalY := _Config.PanelFrontLength;
Radius := _Config.Radius;

IF Radius > (TotalX / 2.0) THEN Radius := TotalX / 2.0; END_IF
IF Radius > (TotalY / 2.0) THEN Radius := TotalY / 2.0; END_IF

IF _ConfigProvider <> 0 THEN
    localConfig := _ConfigProvider.Config;
    Velo := localConfig.CuttingSpeedXY;
ELSE
    Velo := 50.0;
END_IF

// ===================================================
// WYLICZENIE ROZSTAWU OTWORÓW DLA JEDNEGO PANELU
// ===================================================
// Offsety dla szyn (10% z każdego brzegu tak jak we wzorcu)
PanelRailOffsetX := 80;
PanelRailOffsetY := 80;

ExtrusionLengthX := TotalX - (2.0 * PanelRailOffsetX);
ExtrusionLengthY := TotalY - (2.0 * PanelRailOffsetY);

IF NumberOfHolesX > 1 THEN
    HolesSpacingX := (ExtrusionLengthX - (2.0 * HoleDistanceFromEdgeOfRail)) / INT_TO_LREAL(NumberOfHolesX - 1);
ELSE
    HolesSpacingX := 0.0;
END_IF

IF NumberOfHolesY > 1 THEN
    HolesSpacingY := (ExtrusionLengthY - (2.0 * HoleDistanceFromEdgeOfRail)) / INT_TO_LREAL(NumberOfHolesY - 1);
ELSE
    HolesSpacingY := 0.0;
END_IF

// ===================================================
// PRZYPISANIE WSPÓŁRZĘDNYCH OTWORÓW (Po 2 na krawędź)
// ===================================================
holeIdx := 0; 

// 1. Rail Y1 (Lewa)
FOR i := NumberOfHolesY TO 1 BY -1 DO
    holeIdx := holeIdx + 1;
    _HolesDrill[holeIdx].X := LREAL_TO_REAL(PanelRailOffsetX - SomeFixedDimension);
    _HolesDrill[holeIdx].Y := LREAL_TO_REAL(PanelRailOffsetY + HoleDistanceFromEdgeOfRail + ((i - 1) * HolesSpacingY));
END_FOR

// 2. Rail X1 (Dolna)
FOR i := 1 TO NumberOfHolesX DO
    holeIdx := holeIdx + 1;
    _HolesDrill[holeIdx].X := LREAL_TO_REAL(PanelRailOffsetX + HoleDistanceFromEdgeOfRail + ((i - 1) * HolesSpacingX));
    _HolesDrill[holeIdx].Y := LREAL_TO_REAL(PanelRailOffsetY - SomeFixedDimension);
END_FOR

// 3. Rail Y2 (Prawa)
FOR i := 1 TO NumberOfHolesY DO
    holeIdx := holeIdx + 1;
    _HolesDrill[holeIdx].X := LREAL_TO_REAL(PanelRailOffsetX + ExtrusionLengthX + SomeFixedDimension);
    _HolesDrill[holeIdx].Y := LREAL_TO_REAL(PanelRailOffsetY + HoleDistanceFromEdgeOfRail + ((i - 1) * HolesSpacingY));
END_FOR

// 4. Rail X2 (Górna)
FOR i := NumberOfHolesX TO 1 BY -1 DO
    holeIdx := holeIdx + 1;
    _HolesDrill[holeIdx].X := LREAL_TO_REAL(PanelRailOffsetX + HoleDistanceFromEdgeOfRail + ((i - 1) * HolesSpacingX));
    _HolesDrill[holeIdx].Y := LREAL_TO_REAL(PanelRailOffsetY + ExtrusionLengthY + SomeFixedDimension);
END_FOR

_HolesToDrill := holeIdx; // Wynik to dokładnie 8 otworów

// ===================================================
// DEFINICJA KSZTAŁTU (Tylko 1 główny prostokąt)
// ===================================================
_ShapesCount := 1; 

// Zaczynamy na środku PRAWEJ krawędzi
_ShapeStart[1].X := TotalX;
_ShapeStart[1].Y := TotalY / 2.0;

// ============================================
// GENEROWANIE TABELI (Ruch CCW / Lewoskrętnie)
// ============================================
_GeometryWriter.Clear();
_GeometryWriter.EnableTangentialFollowing();

CASE _CurrentShapeIndex OF
    1:
        _GeometryWriter.AddStartPoint(_ShapeStart[1].X, _ShapeStart[1].Y);

        // 1. Prawa krawędź
        _GeometryWriter.AddLine(TotalX, TotalY - Radius, Velo);
        IF Radius > 0 THEN
            _GeometryWriter.AddArc(TotalX - Radius, TotalY, TotalX - Radius, TotalY - Radius, Velo, FALSE);
        END_IF

        // 2. Górna krawędź
        _GeometryWriter.AddLine(Radius, TotalY, Velo);
        IF Radius > 0 THEN
            _GeometryWriter.AddArc(0.0, TotalY - Radius, Radius, TotalY - Radius, Velo, FALSE);
        END_IF

        // 3. Lewa krawędź
        _GeometryWriter.AddLine(0.0, Radius, Velo);
        IF Radius > 0 THEN
            _GeometryWriter.AddArc(Radius, 0.0, Radius, Radius, Velo, FALSE);
        END_IF

        // 4. Dolna krawędź
        _GeometryWriter.AddLine(TotalX - Radius, 0.0, Velo);
        IF Radius > 0 THEN
            _GeometryWriter.AddArc(TotalX, Radius, TotalX - Radius, Radius, Velo, FALSE);
        END_IF

        // Zamknięcie do połowy prawej krawędzi
        _GeometryWriter.AddLine(TotalX, TotalY / 2.0, Velo);

END_CASE

_GeometryWriter.EndTable();

_Busy := FALSE;
_Done := TRUE;
Build := TRUE;
END_METHOD

METHOD PROTECTED CalculateFootprint
VAR_INPUT
END_VAR
_NominalX := _Config.PanelFrontWidth;
_NominalY := _Config.PanelFrontLength;
END_METHOD

PROPERTY ExecutionRoute : E_ExecutionRoute
GET
ExecutionRoute := E_ExecutionRoute.eFeedTable;
END_GET
END_PROPERTY

METHOD FB_init : BOOL
VAR_INPUT
	bInitRetains : BOOL; // if TRUE, the retain variables are initialized (warm start / cold start)
	bInCopyCode : BOOL;  // if TRUE, the instance afterwards gets moved into the copy code (online change)
END_VAR
_Limits.PanelFrontLength.MinVal := 100.0;
_Limits.PanelFrontLength.MaxVal := 2400.0;

_Limits.PanelFrontWidth.MinVal  := 100.0;
_Limits.PanelFrontWidth.MaxVal  := 1200.0;

_Limits.PanelHeight.MinVal      := 0.0;
_Limits.PanelHeight.MaxVal      := 0.0;

_Limits.RailHeightCorrection.MinVal := 0.0;
_Limits.RailHeightCorrection.MaxVal := 0.0;

_Limits.CuttingOverpass.MinVal := 0.0;
_Limits.CuttingOverpass.MaxVal := 50.0;

_Limits.GroovingOverpass.MinVal := 0.0;
_Limits.GroovingOverpass.MaxVal := 50.0;

_Limits.GrooveDepthZ.MinVal := 0.0;
_Limits.GrooveDepthZ.MaxVal := 9.0; 

_Limits.CuttingOverpass.MinVal := 0.0;
_Limits.CuttingOverpass.MaxVal := 50.0;
_Limits.GroovingOverpass.MinVal := 0.0;
_Limits.GroovingOverpass.MaxVal := 50.0;

_Limits.Radius.MinVal := 10.0;     
_Limits.Radius.MaxVal := 600.0;
END_METHOD

END_FUNCTION_BLOCK

// ---- POUs/SAFETY.TcPOU
PROGRAM SAFETY
VAR
END_VAR

END_PROGRAM

// ---- POUs/GantryXYZ/HomingStrategies/FB_Homing_CustomPLC.TcPOU
FUNCTION_BLOCK FB_Homing_CustomPLC EXTENDS FB_Homing_Base
VAR
// =================================================================================
    // IMPORTANT: FOR THIS BLOCK TO WORK, YOU MUST SET THE FOLLOWING IN NC AXIS PARAMETERS:
    // Reference Mode -> 'Application (PLC code)'
    // =================================================================================
    
    fbReadAppReq  : MC_ReadApplicationRequest;
    // fbMcJog       : MC_Jog;
    // fbSetPosition : MC_SetPosition; 
END_VAR

METHOD Abort
VAR_INPUT
END_VAR
SUPER^.Abort();
END_METHOD

METHOD CyclicLogic
CASE nStep OF
    0: // IDLE
    
    10: // READ APPLICATION REQUEST (Placeholder)
        _bBusy := FALSE;
        _bDone := TRUE;
        nStep  := 0;
        
    99: // ERROR HANDLING
        _bBusy    := FALSE;
        _bError   := TRUE;
        _bErrorID := 9999;
        nStep     := 0;
END_CASE
END_METHOD

END_FUNCTION_BLOCK

// ---- POUs/TESTS.TcPOU
PROGRAM TESTS
VAR
//	Test_Extend_TurnsOnValve_And_ReportsExtended 	: FB_Cylinder_Test;
//	Test_MockedExecutor 							: FB_ExecutorCut_Test; 
//	Test_ExecutorGCode  							: FB_ExecutorGCode_Test;
//	Test_GrooveExecutor 							: FB_ExecutorGrooveXY_Test;
//	Test_ExecutorNCITable							: FB_ExecutorNCITable_Test;
//	Test_FeedBuilderRoundedRect 					: FB_FeedBuilderRoundedRect_Test;
//	Test_GantryXYZ									: FB_GantryXYZ_Test;
//	Test_NciChannel            						: FB_NciChannel_Test;
//  Test_NciChannelTangential  						: FB_NciChannelTangential_Test; // Mock Channel
//	Test_RecipeBuilder 								: FB_RecipeBuilder_Test;
//	Test_RecipeFactory 								: FB_RecipeFactory_Test;
//	Test_FB_Exec_Drill_PTP_Test						: FB_Exec_Drill_PTP_Test;
END_VAR

//TcUnit.RUN();

END_PROGRAM

// ---- POUs/TESTS/FB_Cylinder_Test.TcPOU
FUNCTION_BLOCK FB_Cylinder_Test EXTENDS TcUnit.FB_TestSuite
VAR
    Cylinder_ExtendHappy  : FB_Cylinder;
    Cylinder_RetractHappy : FB_Cylinder;
    
    Cylinder_ExtendTime   : FB_Cylinder;
    Cylinder_RetractTime  : FB_Cylinder;
    
    Cylinder_Reset        : FB_Cylinder;
END_VAR

Test_Error_Resets_When_TargetReached();
Test_Extend_Timeout_RaisesError(); 
Test_Extend_TurnsOnValve_And_ReportsExtended();
Test_Retract_Timeout_RaisesError();
Test_Retract_TurnsOffValve_And_ReportsRetracted();

METHOD Test_Error_Resets_When_TargetReached
VAR_INST
    Step : INT := 0;
    TestConfig : ST_Cylinder_Config;
END_VAR


// -------------------------------------------------------------

TEST('Test_Error_Resets_When_TargetReached');
Cylinder_Reset.CyclicLogic();

CASE Step OF
    0: 
        // 1. ARRANGE - Przygotowanie do szybkiego timeoutu
        Cylinder_Reset.Sensor := FALSE; 
        TestConfig := Cylinder_Reset.Config;
        TestConfig.ExtendTime := 0.1; 
        Cylinder_Reset.Config := TestConfig;
        Step := 10;
        
    10: 
        // 2. ACT - Rozkaz i celowe wejście w błąd
        Cylinder_Reset.Extend();
        Step := 20;
        
    20:
        // Czekamy na błąd (symulacja zawieszenia / wolnego powietrza)
        IF Cylinder_Reset.Error THEN
            Step := 30;
        END_IF
        
    30:
        // 3. ACT - Błąd trwa, ale nagle sprzęt fizycznie osiąga cel (czujnik łapie!)
        Cylinder_Reset.Sensor := TRUE;
        Step := 40;
        
    40:
        // 4. ASSERT - Siłownik powinien zgasić błąd na podstawie czujnika i flagi Request
        AssertFalse(Condition := Cylinder_Reset.Error, 
                    Message := 'Blad timeoutu nie zresetowal sie pomimo osiagniecia celu!');
                    
        AssertTrue(Condition := Cylinder_Reset.Extended, 
                   Message := 'Pomimo bledu, silownik nie zglosil Extended po zlapaniu czujnika!');
                   
        TEST_FINISHED();
END_CASE
END_METHOD

METHOD Test_Extend_Timeout_RaisesError
VAR_INST
    Step : INT := 0;
    TestConfig : ST_Cylinder_Config;
END_VAR


// Rejestrujemy nowy test
TEST('Test_Extend_Timeout_RaisesError');

// Cykl PLC
Cylinder_ExtendTime.CyclicLogic();

CASE Step OF
    0:
        // 1. ARRANGE
        Cylinder_ExtendTime.Sensor := FALSE; // Czujnik nie widzi siłownika
        
        // Ustawiamy bardzo krótki czas wysuwu, żeby test w TcUnit wykonał się błyskawicznie (0.1 sekundy)
        TestConfig := Cylinder_ExtendTime.Config;
        TestConfig.ExtendTime := 0.1; 
        Cylinder_ExtendTime.Config := TestConfig;
        
        Step := 10;
        
    10:
        // 2. ACT - Rozkaz wysunięcia
        Cylinder_ExtendTime.Extend();
        Step := 20;
        
    20:
        // 3. ACT & ASSERT - Czekamy na błąd
        // Nie aktywujemy czujnika! Zostawiamy go na FALSE.
        // Jeśli timer minie (0.1s), siłownik powinien zgłosić Error.
        
        IF Cylinder_ExtendTime.Error THEN
            // Sprawdzamy, czy podniósł się alarm z odpowiednim ID (1)
AssertEquals_UDINT(Expected := 2,  // Zmieniamy na 2, bo to jest faktyczne ID tego błędu w systemie
                   Actual := Cylinder_ExtendTime.ErrorID, 
                   Message := 'Zle ID bledu dla timeoutu siownika!');
                               
            TEST_FINISHED(); // Test udany - kod poprawnie wykrył awarię!
        END_IF
        
        // Zabezpieczenie testu: jeśli coś nie działa w kodzie i Error nigdy nie nastąpi,
        // TcUnit ma własny watchdog i po kilku sekundach uwali ten test jako "Timeout".
END_CASE
END_METHOD

METHOD Test_Extend_TurnsOnValve_And_ReportsExtended
VAR_INST
    Step : INT := 0;
    TestConfig : ST_Cylinder_Config; // Zmienna lokalna na konfigurację
END_VAR

// To musi być wywołane co cykl, żeby TcUnit śledził stan testu
TEST('Test_Extend_TurnsOnValve_And_ReportsExtended');

// Symulujemy cykl pracy PLC dla siłownika
Cylinder_ExtendHappy.CyclicLogic();

CASE Step OF
    0: 
        // 1. ARRANGE - Ustawiamy warunki początkowe
        Cylinder_ExtendHappy.Sensor := FALSE; // Udajemy, że czujnik nie widzi siłownika
        
        // Zgrywamy config, nadpisujemy i wstrzykujemy przez nowe Property
        TestConfig := Cylinder_ExtendHappy.Config;
        TestConfig.ExtendTime := 2.0; 
        Cylinder_ExtendHappy.Config := TestConfig;
        
        Step := 10;
        
    10: 
        // 2. ACT - Wysyłamy komendę wysunięcia
        Cylinder_ExtendHappy.Extend();
        
        // Przechodzimy do kolejnego kroku, żeby dać szansę CyclicLogic() na reakcję
        Step := 20;
        
    20:
        // 3. ASSERT - Krok pośredni
        // Skoro w poprzednim cyklu daliśmy Extend(), zawór powinien być już otwarty
        AssertTrue(Condition := Cylinder_ExtendHappy.Valve, 
                   Message := 'Zawor wysuwu (CylinderValveCutX) nie zostal wysterowany!');
                   
        // 4. ACT - Symulujemy, że fizyczny siłownik dojechał do końca i czujnik łapie
        Cylinder_ExtendHappy.Sensor := TRUE;
        
        Step := 30;
        
    30:
        // 5. ASSERT - Weryfikacja końcowa
        AssertTrue(Condition := Cylinder_ExtendHappy.Extended, 
                   Message := 'Cylinder nie zaraportowal stanu Extended po aktywacji czujnika!');
                   
        // Zakańczamy test
        TEST_FINISHED();
        
END_CASE
END_METHOD

METHOD Test_Retract_Timeout_RaisesError
VAR_INST
    Step : INT := 0;
    TestConfig : ST_Cylinder_Config;
END_VAR


// -------------------------------------------------------------

TEST('Test_Retract_Timeout_RaisesError');
Cylinder_RetractTime.CyclicLogic();

CASE Step OF
    0:
        // 1. ARRANGE - Cylinder jest wysunięty
        Cylinder_RetractTime.Sensor := TRUE; 
        
        TestConfig := Cylinder_RetractTime.Config;
        TestConfig.RetractTime := 0.1; // Szybki timeout
        Cylinder_RetractTime.Config := TestConfig;
        
        Step := 10;
        
    10:
        // 2. ACT
        Cylinder_RetractTime.Retract();
        Step := 20;
        
    20:
        // 3. ASSERT - Czekamy na błąd, NIE zmieniamy stanu czujnika!
        IF Cylinder_RetractTime.Error THEN
            AssertTrue(Condition := TRUE, Message := 'Ten Assert zawsze przechodzi, potwierdza Error');
            TEST_FINISHED();
        END_IF
END_CASE
END_METHOD

METHOD Test_Retract_TurnsOffValve_And_ReportsRetracted
VAR_INST
    Step : INT := 0;
    TestConfig : ST_Cylinder_Config;
END_VAR


// -------------------------------------------------------------

TEST('Test_Retract_TurnsOffValve_And_ReportsRetracted');
Cylinder_RetractHappy.CyclicLogic();

CASE Step OF
    0: 
        // 1. ARRANGE - Ustawiamy warunki początkowe (Cylinder jest wysunięty)
        Cylinder_RetractHappy.Sensor := TRUE; 
        
        TestConfig := Cylinder_RetractHappy.Config;
        TestConfig.RetractTime := 2.0; 
        Cylinder_RetractHappy.Config := TestConfig;
        
        Step := 10;
        
    10: 
        // 2. ACT - Wysyłamy komendę wsunięcia
        Cylinder_RetractHappy.Retract();
        Step := 20;
        
    20:
        // 3. ASSERT - Krok pośredni (Zawór musi się natychmiast wyłączyć)
        AssertFalse(Condition := Cylinder_RetractHappy.Valve, 
                    Message := 'Zawor nie zostal wylaczony przy komendzie chowania!');
                    
        // 4. ACT - Symulujemy zjechanie z czujnika (powrót)
        Cylinder_RetractHappy.Sensor := FALSE;
        Step := 30;
        
